	        // Check which specific status changed, prepare code, change state and write new status into the old one.
	        IF (#i_UDT_ArmDiverterStatus.Specific.TimeoutError <> #s_UDT_ArmDiverterOldStatus.Specific.TimeoutError AND NOT #sx_SendAllProcedure)
	            OR (#sx_SendAllProcedure AND #ii_ErrorNumber = 0)
	        THEN
	            #sdi_Code := "DB_MFC_ErrorCode".ArmDiverter.TimeoutError;
	            #si_State := BOOL_TO_INT(#i_UDT_ArmDiverterStatus.Specific.TimeoutError);
	            #s_UDT_ArmDiverterOldStatus.Specific.TimeoutError := #i_UDT_ArmDiverterStatus.Specific.TimeoutError;
	            #sx_ItemErrorMessageReq := TRUE;
	            #ii_ErrorNumber += 1;
	        ELSIF (#i_UDT_ArmDiverterStatus.Specific.LimitHomeError <> #s_UDT_ArmDiverterOldStatus.Specific.LimitHomeError AND NOT #sx_SendAllProcedure)
	            OR (#sx_SendAllProcedure AND #ii_ErrorNumber = 1)
	        THEN
	            #sdi_Code := "DB_MFC_ErrorCode".ArmDiverter.LimitHomeError;
	            #si_State := BOOL_TO_INT(#i_UDT_ArmDiverterStatus.Specific.LimitHomeError);
	            #s_UDT_ArmDiverterOldStatus.Specific.LimitHomeError := #i_UDT_ArmDiverterStatus.Specific.LimitHomeError;
	            #sx_ItemErrorMessageReq := TRUE;
	            #ii_ErrorNumber += 1;
	        ELSIF (#i_UDT_ArmDiverterStatus.Specific.LimitDivertError <> #s_UDT_ArmDiverterOldStatus.Specific.LimitDivertError AND NOT #sx_SendAllProcedure)
	            OR (#sx_SendAllProcedure AND #ii_ErrorNumber = 2)
	        THEN
	            #sdi_Code := "DB_MFC_ErrorCode".ArmDiverter.LimitDivertError;
	            #si_State := BOOL_TO_INT(#i_UDT_ArmDiverterStatus.Specific.LimitDivertError);
	            #s_UDT_ArmDiverterOldStatus.Specific.LimitDivertError := #i_UDT_ArmDiverterStatus.Specific.LimitDivertError;
	            #sx_ItemErrorMessageReq := TRUE;
	            #ii_ErrorNumber += 1;
	        ELSIF (#i_UDT_ArmDiverterStatus.Specific.PXHomeError <> #s_UDT_ArmDiverterOldStatus.Specific.PXHomeError AND NOT #sx_SendAllProcedure)
	            OR (#sx_SendAllProcedure AND #ii_ErrorNumber = 3)
	        THEN
	            #sdi_Code := "DB_MFC_ErrorCode".ArmDiverter.PXHomeError;
	            #si_State := BOOL_TO_INT(#i_UDT_ArmDiverterStatus.Specific.PXHomeError);
	            #s_UDT_ArmDiverterOldStatus.Specific.PXHomeError := #i_UDT_ArmDiverterStatus.Specific.PXHomeError;
	            #sx_ItemErrorMessageReq := TRUE;
	            #ii_ErrorNumber += 1;
	        ELSIF (#i_UDT_ArmDiverterStatus.Specific.PXDivertError <> #s_UDT_ArmDiverterOldStatus.Specific.PXDivertError AND NOT #sx_SendAllProcedure)
	            OR (#sx_SendAllProcedure AND #ii_ErrorNumber = 4)
	        THEN
	            #sdi_Code := "DB_MFC_ErrorCode".ArmDiverter.PXDivertError;
	            #si_State := BOOL_TO_INT(#i_UDT_ArmDiverterStatus.Specific.PXDivertError);
	            #s_UDT_ArmDiverterOldStatus.Specific.PXDivertError := #i_UDT_ArmDiverterStatus.Specific.PXDivertError;
	            #sx_ItemErrorMessageReq := TRUE;
	            #ii_ErrorNumber += 1;
	        ELSIF (#i_UDT_ArmDiverterStatus.Specific.AtHomePosition <> #s_UDT_ArmDiverterOldStatus.Specific.AtHomePosition AND NOT #sx_SendAllProcedure)
	            OR (#sx_SendAllProcedure AND #ii_ErrorNumber = 5)
	        THEN
	            #sdi_Code := "DB_MFC_ErrorCode".ArmDiverter.AtHomePosition;
	            #si_State := BOOL_TO_INT(#i_UDT_ArmDiverterStatus.Specific.AtHomePosition);
	            #s_UDT_ArmDiverterOldStatus.Specific.AtHomePosition := #i_UDT_ArmDiverterStatus.Specific.AtHomePosition;
	            #sx_ItemErrorMessageReq := TRUE;
	            #ii_ErrorNumber += 1;
	        ELSIF (#i_UDT_ArmDiverterStatus.Specific.AtDivertPosition <> #s_UDT_ArmDiverterOldStatus.Specific.AtDivertPosition AND NOT #sx_SendAllProcedure)
	            OR (#sx_SendAllProcedure AND #ii_ErrorNumber = 6)
	        THEN
	            #sdi_Code := "DB_MFC_ErrorCode".ArmDiverter.AtDivertPosition;
	            #si_State := BOOL_TO_INT(#i_UDT_ArmDiverterStatus.Specific.AtDivertPosition);
	            #s_UDT_ArmDiverterOldStatus.Specific.AtDivertPosition := #i_UDT_ArmDiverterStatus.Specific.AtDivertPosition;
	            #sx_ItemErrorMessageReq := TRUE;
	            #ii_ErrorNumber += 1;
	        ELSIF (#i_UDT_ArmDiverterStatus.Specific.ReferencError <> #s_UDT_ArmDiverterOldStatus.Specific.ReferencError AND NOT #sx_SendAllProcedure)
	            OR (#sx_SendAllProcedure AND #ii_ErrorNumber = 7)
	        THEN
	            #sdi_Code := "DB_MFC_ErrorCode".ArmDiverter.ReferencError;
	            #si_State := BOOL_TO_INT(#i_UDT_ArmDiverterStatus.Specific.ReferencError);
	            #s_UDT_ArmDiverterOldStatus.Specific.ReferencError := #i_UDT_ArmDiverterStatus.Specific.ReferencError;
	            #sx_ItemErrorMessageReq := TRUE;
	            #ii_ErrorNumber += 1;
	        ELSIF (#i_UDT_ArmDiverterStatus.Specific.ParcelDivertError <> #s_UDT_ArmDiverterOldStatus.Specific.ParcelDivertError AND NOT #sx_SendAllProcedure)
	            OR (#sx_SendAllProcedure AND #ii_ErrorNumber = 8)
	        THEN
	            #sdi_Code := "DB_MFC_ErrorCode".ArmDiverter.ParcelDivertError;
	            #si_State := BOOL_TO_INT(#i_UDT_ArmDiverterStatus.Specific.ParcelDivertError);
	            #s_UDT_ArmDiverterOldStatus.Specific.ParcelDivertError := #i_UDT_ArmDiverterStatus.Specific.ParcelDivertError;
	            #sx_ItemErrorMessageReq := TRUE;
	            #sx_SendAllProcedure := FALSE;
	        END_IF;
	    END_IF;
	END_REGION

	REGION 4 - Write message components to the item error structure

	    #s_UDT_ItemError.ItemNumber := #i_UDT_EquipmentNumber;
	    #s_UDT_ItemError.Error := #sdi_Code;
	    #s_UDT_ItemError.State := #si_State;
	    #s_UDT_ItemError.Masked := 1;

	END_REGION

	REGION 5 - Write message components to the item status structure

	    #s_UDT_ItemStatus.Group := #i_UDT_EquipmentNumber.Group;
	    #s_UDT_ItemStatus.Node := #i_UDT_EquipmentNumber.Node;
	    #s_UDT_ItemStatus.Status := #si_ItemStatus;

	END_REGION

	REGION 6 - Prepare messages to the MFC

	    // If item error message required signal is set, prepare the item error message.
	    IF (#sx_ItemErrorMessageReq)
	    THEN
	        #s_FB_ItemError(i_UDT_ItemErrorBody := #s_UDT_ItemError,
	                        ii_MessageGroup := 1,
	                        ix_FlagRetry := FALSE,
	                        idi_TimeSpan := 0,
	                        qx_Error => #sx_ItemErrorBlockError,
	                        qx_Warning => #sx_ItemErrorBlockWarning,
	                        iq_UDT_FifoHeader := #iq_UDT_FifoHeader,
	                        iqs_FifoData := #iqs_FifoData,
	                        iqdi_MessageSequenceNumber := #iqdi_MessageSequenceNumber);
	    END_IF;

	    // If item status message required signal is set, prepare the item error message.
	    IF (#sx_ItemStatusMessageReq)
	    THEN
	        #s_FB_ItemStatus(i_UDT_ItemStatusBody := #s_UDT_ItemStatus,
	                         ii_MessageGroup := 1,
	                         ix_FlagRetry := FALSE,
	                         idi_TimeSpan := 0,
	                         qx_Error => #sx_ItemStatusBlockError,
	                         qx_Warning => #sx_ItemStatusBlockWarning,
	                         iq_UDT_FifoHeader := #iq_UDT_FifoHeader,
	                         iqs_FifoData := #iqs_FifoData,
	                         iqdi_MessageSequenceNumber := #iqdi_MessageSequenceNumber);
	    END_IF;

	END_REGION

	REGION 7 - Write outputs

	    // Prepare collective output error.
	    #qx_Error :=
	    #sx_ItemErrorBlockError
	    OR #sx_ItemStatusBlockError
	    OR #sx_FIFOError;

	    // Prepare collective output warning.
	    #qx_Warning :=
	    #sx_ItemErrorBlockWarning
	    OR #sx_ItemStatusBlockWarning
	    OR #sx_FIFOWarning;

	END_REGION




END_FUNCTION_BLOCK

FUNCTION_BLOCK "FB_MFC_Visu_TCPIPSend"
TITLE = FB_TCPIPSend
{ S7_Optimized_Access := 'TRUE' }
AUTHOR : MHSE
FAMILY : Communication
VERSION : 2.0
// ATTRIBUTES
// AUTO_NUMBER = True
// BLOCK_NUMBER = 162
// END_ATTRIBUTES
//Function block to send data from TCPIP.
   VAR_INPUT
      i_UDT_Connection { ExternalAccessible := 'False'; ExternalVisible := 'False'; ExternalWritable := 'False'} : "UDT_Connection";   // Connection parameters
      ii_HeaderLength { ExternalAccessible := 'False'; ExternalVisible := 'False'; ExternalWritable := 'False'} : Int;   // Message header length
      ii_BodyLengthPosition { ExternalAccessible := 'False'; ExternalVisible := 'False'; ExternalWritable := 'False'} : Int;   // Position in header where message body length value starts
      ix_EnableSend { ExternalAccessible := 'False'; ExternalVisible := 'False'; ExternalWritable := 'False'} : Bool;   // TRUE when send is enable
   END_VAR

   VAR_OUTPUT
      qx_Error { ExternalAccessible := 'False'; ExternalVisible := 'False'; ExternalWritable := 'False'} : Bool;   // TRUE when collective block error occurred
      qx_Warning { ExternalAccessible := 'False'; ExternalVisible := 'False'; ExternalWritable := 'False'} : Bool;   // TRUE when collective block warning occurred
   END_VAR

   VAR_IN_OUT
      iq_UDT_FifoLowHeader : "UDT_FifoHeader";   // Low priority FIFO header
      iqs_FifoLowData : Variant;   // Low priority FIFO data
      iq_UDT_FifoMediumHeader : "UDT_FifoHeader";   // Medium priority FIFO header
      iqs_FifoMediumData : Variant;   // Medium priority FIFO data
      iq_UDT_FifoHighHeader : "UDT_FifoHeader";   // High priority FIFO header
      iqs_FifoHighData : Variant;   // High priority FIFO data
   END_VAR

   VAR
      s_FB_TSEND {InstructionName := 'TSEND'; LibVersion := '4.0'; ExternalAccessible := 'False'; ExternalVisible := 'False'; ExternalWritable := 'False'; S7_SetPoint := 'False'} : TSEND;   // Siemens "TSEND" block - to send the data over TCPIP socket
      s_UDT_MessageArray { ExternalAccessible := 'False'; ExternalVisible := 'False'; ExternalWritable := 'False'; S7_SetPoint := 'False'} : "UDT_MessageV2";   // Message
      ss_TSEND { ExternalAccessible := 'False'; ExternalVisible := 'False'; ExternalWritable := 'False'} : Struct   // TSEND block structure
         Status { ExternalAccessible := 'False'; ExternalVisible := 'False'; ExternalWritable := 'False'} : Word;   //    TSEND - Status
         Request { ExternalAccessible := 'False'; ExternalVisible := 'False'; ExternalWritable := 'False'} : Bool;   //    TSEND - Request
         Busy { ExternalAccessible := 'False'; ExternalVisible := 'False'; ExternalWritable := 'False'} : Bool;   //    TSEND - Busy
         Done { ExternalAccessible := 'False'; ExternalVisible := 'False'; ExternalWritable := 'False'} : Bool;   //    TSEND - Done
         Error { ExternalAccessible := 'False'; ExternalVisible := 'False'; ExternalWritable := 'False'} : Bool;   //    TSEND - Error
      END_STRUCT;
      ss_Status { ExternalAccessible := 'False'; ExternalVisible := 'False'; ExternalWritable := 'False'} : Struct   // Status structure
         FIFOLowPriorityStatus { ExternalAccessible := 'False'; ExternalVisible := 'False'; ExternalWritable := 'False'} : "UDT_FifoStatus";
         FIFOMedPriorityStatus { ExternalAccessible := 'False'; ExternalVisible := 'False'; ExternalWritable := 'False'} : "UDT_FifoStatus";
         FIFOHighPriorityStatus { ExternalAccessible := 'False'; ExternalVisible := 'False'; ExternalWritable := 'False'} : "UDT_FifoStatus";
         FIFOLowPriorityError { ExternalAccessible := 'False'; ExternalVisible := 'False'; ExternalWritable := 'False'} : Bool;   // FIFO low priority error
         FIFOLowPriorityWarning { ExternalAccessible := 'False'; ExternalVisible := 'False'; ExternalWritable := 'False'} : Bool;   // FIFO low priority warning
         FIFOMedPriorityError { ExternalAccessible := 'False'; ExternalVisible := 'False'; ExternalWritable := 'False'} : Bool;   // FIFO medium priority error
         FIFOMedPriorityWarning { ExternalAccessible := 'False'; ExternalVisible := 'False'; ExternalWritable := 'False'} : Bool;   // FIFO medium priority warning
         FIFOHighPriorityError { ExternalAccessible := 'False'; ExternalVisible := 'False'; ExternalWritable := 'False'} : Bool;   // FIFO high priority error
         FIFOHighPriorityWarning { ExternalAccessible := 'False'; ExternalVisible := 'False'; ExternalWritable := 'False'} : Bool;   // FIFO high priority warning
         SendError { ExternalAccessible := 'False'; ExternalVisible := 'False'; ExternalWritable := 'False'} : Bool;   // Send operation error
      END_STRUCT;
      sw_BodyLength { ExternalAccessible := 'False'; ExternalVisible := 'False'; ExternalWritable := 'False'} : Word;   // Message body length
      si_MessageLength { ExternalAccessible := 'False'; ExternalVisible := 'False'; ExternalWritable := 'False'} : Int;   // Message length
      sx_MessageReady { ExternalAccessible := 'False'; ExternalVisible := 'False'; ExternalWritable := 'False'} : Bool;   // Message is ready to send
      sx_MessageRead { ExternalAccessible := 'False'; ExternalVisible := 'False'; ExternalWritable := 'False'} : Bool;   // Message has been read
      sx_MessageReadRequest { ExternalAccessible := 'False'; ExternalVisible := 'False'; ExternalWritable := 'False'} : Bool;   // Request to read message
      sx_FIFOError { ExternalAccessible := 'False'; ExternalVisible := 'False'; ExternalWritable := 'False'} : Bool;   // Summary FIFO error
   END_VAR


BEGIN
	(*
	----------------------------------------------------------------------------------------
	|                                                                                      |
	|  Copyright  2023             FORTNA Europe BV                                        |
	|  All Rights Reserved         Netherlands                                             |
	|                                                                                      |
	----------------------------------------------------------------------------------------
	Version history:
	Date        | Version   | Author       | Remark
	----------------------------------------------------------------------------------------
	24/10/2019  | 3.0       | L.Klar       | Initial version
	12/03/2020  | 3.1       | M.Kurpiers   | Adapting reviews
	16/01/2023  | 4.0       | S. Nikodem   | Release TIA 17 | DHL Munich 2023
	13/03/2023  | 4.1       | S. Nieswiec  | Updated for new Baseline
	*)

	REGION 1 – Update FIFO header status bits

	    // Mode 'S' - High priority FIFO register status update.
	    "FC_Fifo"(ic_Mode := 'S',
	              qUDT_Status => #ss_Status.FIFOHighPriorityStatus,
	              qx_Error => #ss_Status.FIFOHighPriorityError,
	              qx_Warning => #ss_Status.FIFOHighPriorityWarning,
	              iqv_Data := #s_UDT_MessageArray,
	              iqUDT_FifoHeader := #iq_UDT_FifoHighHeader,
	              iqv_DataBuffer := #iqs_FifoHighData);

	    // Mode 'S' - Medium priority FIFO register status update.
	    "FC_Fifo"(ic_Mode := 'S',
	              qUDT_Status => #ss_Status.FIFOMedPriorityStatus,
	              qx_Error => #ss_Status.FIFOMedPriorityError,
	              qx_Warning => #ss_Status.FIFOMedPriorityWarning,
	              iqv_Data := #s_UDT_MessageArray,
	              iqUDT_FifoHeader := #iq_UDT_FifoMediumHeader,
	              iqv_DataBuffer := #iqs_FifoMediumData);

	    // Mode 'S' - Low priority FIFO register status update.
	    "FC_Fifo"(ic_Mode := 'S',
	              qUDT_Status => #ss_Status.FIFOLowPriorityStatus,
	              qx_Error => #ss_Status.FIFOLowPriorityError,
	              qx_Warning => #ss_Status.FIFOLowPriorityWarning,
	              iqv_Data := #s_UDT_MessageArray,
	              iqUDT_FifoHeader := #iq_UDT_FifoLowHeader,
	              iqv_DataBuffer := #iqs_FifoLowData);

	END_REGION

	REGION 2 – FIFO header summary error

	    #sx_FIFOError :=
	    #ss_Status.FIFOHighPriorityError
	    OR #ss_Status.FIFOMedPriorityError
	    OR #ss_Status.FIFOLowPriorityError;

	END_REGION

	REGION 3 – FIFO Read request

	    #sx_MessageReadRequest :=
	    #ix_EnableSend
	    AND NOT #sx_FIFOError
	    AND NOT #ss_TSEND.Error
	    AND #ss_TSEND.Status = 16#7000;

	END_REGION

	REGION 4 – Read the message from high priority FIFO data buffer

	    IF #sx_MessageReadRequest
	        AND NOT #iq_UDT_FifoHighHeader.Status.Empty
	        AND NOT #sx_MessageRead
	    THEN
	        // Mode 'R' - Read high priority FIFO record.
	        "FC_Fifo"(ic_Mode := 'R',
	                  qUDT_Status => #ss_Status.FIFOHighPriorityStatus,
	                  qx_Error => #ss_Status.FIFOHighPriorityError,
	                  qx_Warning => #ss_Status.FIFOHighPriorityWarning,
	                  iqv_Data := #s_UDT_MessageArray,
	                  iqUDT_FifoHeader := #iq_UDT_FifoHighHeader,
	                  iqv_DataBuffer := #iqs_FifoHighData);

	        #sx_MessageRead := TRUE;
	    END_IF;

	END_REGION

	REGION 5 – Read the message from medium priority FIFO data buffer

	    IF #sx_MessageReadRequest
	        AND #iq_UDT_FifoHighHeader.Status.Empty
	        AND NOT #iq_UDT_FifoMediumHeader.Status.Empty
	        AND NOT #sx_MessageRead
	    THEN
	        // Mode 'R' - Read medium priority FIFO record.
	        "FC_Fifo"(ic_Mode := 'R',
	                  qUDT_Status => #ss_Status.FIFOMedPriorityStatus,
	                  qx_Error => #ss_Status.FIFOMedPriorityError,
	                  qx_Warning => #ss_Status.FIFOMedPriorityWarning,
	                  iqv_Data := #s_UDT_MessageArray,
	                  iqUDT_FifoHeader := #iq_UDT_FifoMediumHeader,
	                  iqv_DataBuffer := #iqs_FifoMediumData);

	        #sx_MessageRead := TRUE;
	    END_IF;

	END_REGION

	REGION 6 – Read the message from low priority FIFO data buffer

	    IF #sx_MessageReadRequest
	        AND #iq_UDT_FifoHighHeader.Status.Empty
	        AND #iq_UDT_FifoMediumHeader.Status.Empty
	        AND NOT #iq_UDT_FifoLowHeader.Status.Empty
	        AND NOT #sx_MessageRead
	    THEN
	        #sx_MessageRead := TRUE;

	        // Mode 'R' - Read low priority FIFO record.
	        "FC_Fifo"(ic_Mode := 'R',
	                  qUDT_Status => #ss_Status.FIFOLowPriorityStatus,
	                  qx_Error => #ss_Status.FIFOLowPriorityError,
	                  qx_Warning => #ss_Status.FIFOLowPriorityWarning,
	                  iqv_Data := #s_UDT_MessageArray,
	                  iqUDT_FifoHeader := #iq_UDT_FifoLowHeader,
	                  iqv_DataBuffer := #iqs_FifoLowData);
	    END_IF;

	END_REGION

	REGION 7 – Message length

	    // Measuring the length of a read message.
	    IF #sx_MessageRead
	        AND NOT #sx_MessageReady
	    THEN
	        // Initialize the message length.
	        #si_MessageLength := 0;

	        // Get the length of the message by extracting the body length from the message header.
	        #sw_BodyLength := #s_UDT_MessageArray.Bytes[#ii_BodyLengthPosition];
	        #si_MessageLength := WORD_TO_INT(IN := SHL(IN := #sw_BodyLength, N := 8)) + BYTE_TO_INT(#s_UDT_MessageArray.Bytes[#ii_BodyLengthPosition + 1]) + #ii_HeaderLength;
	        #sx_MessageReady := TRUE;
	    END_IF;

	END_REGION

	REGION 8 – Send request

	    IF #sx_MessageRead
	        AND #sx_MessageReady
	    THEN
	        #ss_TSEND.Request := TRUE;
	    END_IF;

	END_REGION

	REGION 9 – Send data

	    #s_FB_TSEND(REQ := #ss_TSEND.Request,
	                ID := #i_UDT_Connection.ID,
	                LEN := INT_TO_UDINT(#si_MessageLength),
	                DONE => #ss_TSEND.Done,
	                BUSY => #ss_TSEND.Busy,
	                ERROR => #ss_TSEND.Error,
	                STATUS => #ss_TSEND.Status,
	                DATA := #s_UDT_MessageArray);

	    // Reset send request, message read and ready bits.
	    IF #ss_TSEND.Request
	        AND NOT #ss_TSEND.Busy
	        AND (#ss_TSEND.Done
	        OR #ss_TSEND.Status = 16#7000)
	    THEN
	        #ss_TSEND.Request := FALSE;
	        #sx_MessageRead := FALSE;
	        #sx_MessageReady := FALSE;
	    END_IF;

	    // Reset send error and TSEND status after correctly sent message.
	    IF #ss_TSEND.Done
	    THEN
	        #ss_Status.SendError := FALSE;
	    END_IF;

	    // Set send error and TSEND status if error occured.
	    IF #ss_TSEND.Error
	    THEN
	        #ss_Status.SendError := TRUE;
	    END_IF;

	END_REGION

	REGION 10 – Status

	    // Parametrization collective error output.
	    #qx_Error :=
	    #sx_FIFOError
	    OR #ss_Status.SendError;

	    // Parametrization collective warning output.
	    #qx_Warning :=
	    #ss_Status.FIFOHighPriorityWarning
	    OR #ss_Status.FIFOMedPriorityWarning
	    OR #ss_Status.FIFOLowPriorityWarning;

	END_REGION
END_FUNCTION_BLOCK

FUNCTION_BLOCK "FB_MFC_Visu_Conveyor_Status"
{ S7_Optimized_Access := 'TRUE' }
VERSION : 0.1
// ATTRIBUTES
// AUTO_NUMBER = True
// BLOCK_NUMBER = 141
// END_ATTRIBUTES
   VAR_INPUT
      ix_SendAllErrorsState { ExternalAccessible := 'False'; ExternalVisible := 'False'; ExternalWritable := 'False'} : Bool;   // True - update all the messages
      ix_MFCConnected { ExternalAccessible := 'False'; ExternalVisible := 'False'; ExternalWritable := 'False'} : Bool;   // True - A connection to the MFC has been established
      ix_CollectiveReset { ExternalAccessible := 'False'; ExternalVisible := 'False'; ExternalWritable := 'False'} : Bool;   // True - Collective reset command of all system controls
      i_UDT_MaintenanceCounterConfiguration { ExternalAccessible := 'False'; ExternalVisible := 'False'; ExternalWritable := 'False'} : "UDT_MaintenanceCounterConfiguration" := (86400, 10000000, 100);   // Maintenance counter configuration
      i_UDT_ConveyorInterface { ExternalAccessible := 'False'; ExternalVisible := 'False'; ExternalWritable := 'False'} : "UDT_ConveyorInterface";   // Input conveyor interface structrue
      i_UDT_ConveyorStatus { ExternalAccessible := 'False'; ExternalVisible := 'False'; ExternalWritable := 'False'} : "UDT_ConveyorStatus";   // Input Conveyor status structure
      i_UDT_EquipmentNumber { ExternalAccessible := 'False'; ExternalVisible := 'False'; ExternalWritable := 'False'} : "UDT_EquipmentNumber";   // Item number
   END_VAR

   VAR_OUTPUT
      qx_Error { ExternalAccessible := 'False'; ExternalVisible := 'False'; ExternalWritable := 'False'} : Bool;   // Block error
      qx_Warning { ExternalAccessible := 'False'; ExternalVisible := 'False'; ExternalWritable := 'False'} : Bool;   // Block warning
   END_VAR

   VAR_IN_OUT
      iq_UDT_FifoHeader : "UDT_FifoHeader";   // FIFO header
      iqs_FifoData : Array[*] of "UDT_MessageV2";   // FIFO data buffer
      iqdi_MessageSequenceNumber { ExternalAccessible := 'False'; ExternalVisible := 'False'; ExternalWritable := 'False'} : DInt;   // Message number
   END_VAR

   VAR
      s_FB_ItemError { ExternalAccessible := 'False'; ExternalVisible := 'False'; ExternalWritable := 'False'; S7_SetPoint := 'False'} : "FB_ItemError";   // Item error block's instance
      s_FB_ItemStatus { ExternalAccessible := 'False'; ExternalVisible := 'False'; ExternalWritable := 'False'; S7_SetPoint := 'False'} : "FB_ItemStatus";   // Item status block's instance
      s_FB_MaintenanceCounter { ExternalAccessible := 'False'; ExternalVisible := 'False'; ExternalWritable := 'False'; S7_SetPoint := 'False'} : "FB_MaintenanceCounter";   // Maintenence counter message block instance
      s_UDT_ItemError { ExternalAccessible := 'False'; ExternalVisible := 'False'; ExternalWritable := 'False'; S7_SetPoint := 'False'} : "UDT_ItemError";   // Item error message body structure
      s_UDT_ItemStatus { ExternalAccessible := 'False'; ExternalVisible := 'False'; ExternalWritable := 'False'; S7_SetPoint := 'False'} : "UDT_ItemStatus";   // Item status message body structure
      s_UDT_Message { ExternalAccessible := 'False'; ExternalVisible := 'False'; ExternalWritable := 'False'; S7_SetPoint := 'False'} : "UDT_BytesMessage";   // Message
      s_UDT_ConveyorOld { ExternalAccessible := 'False'; ExternalVisible := 'False'; ExternalWritable := 'False'; S7_SetPoint := 'False'} : "UDT_ConveyorStatus";   // Conveyor old status structure
      s_UDT_ConveyorInterfaceOld { ExternalAccessible := 'False'; ExternalVisible := 'False'; ExternalWritable := 'False'; S7_SetPoint := 'False'} : "UDT_ConveyorInterface";   // Conveyor old interface structure
      s_UDT_FIFOStatus { ExternalAccessible := 'False'; ExternalVisible := 'False'; ExternalWritable := 'False'; S7_SetPoint := 'False'} : "UDT_FifoStatus";   // FIFO status structure
      ss_FIFOStatus { ExternalAccessible := 'False'; ExternalVisible := 'False'; ExternalWritable := 'False'; S7_SetPoint := 'False'} : "UDT_FifoStatus";   // Status structure
      s_R_TRIG_ConveyorStart {InstructionName := 'R_TRIG'; LibVersion := '1.0'; ExternalAccessible := 'False'; ExternalVisible := 'False'; ExternalWritable := 'False'; S7_SetPoint := 'False'} : R_TRIG;   // Rising edge trigger Conveyor start
      s_R_TRIG_Connection {InstructionName := 'R_TRIG'; LibVersion := '1.0'; ExternalAccessible := 'False'; ExternalVisible := 'False'; ExternalWritable := 'False'; S7_SetPoint := 'False'} : R_TRIG;   // Rising edge trigger connection reastablished
      s_F_TRIG_ConveyorStop {InstructionName := 'F_TRIG'; LibVersion := '1.0'; ExternalAccessible := 'False'; ExternalVisible := 'False'; ExternalWritable := 'False'; S7_SetPoint := 'False'} : F_TRIG;   // Falling edge trigger Conveyor stop
      s_F_TRIG_SendAllErrors {InstructionName := 'F_TRIG'; LibVersion := '1.0'; ExternalAccessible := 'False'; ExternalVisible := 'False'; ExternalWritable := 'False'; S7_SetPoint := 'False'} : F_TRIG;   // Falling edge trigger from signal send all errors
      slr_RunningTimeMS { ExternalAccessible := 'False'; ExternalVisible := 'False'; ExternalWritable := 'False'} : LReal;   // Conveyor running time [ms]
      sdi_DistanceTraveled { ExternalAccessible := 'False'; ExternalVisible := 'False'; ExternalWritable := 'False'} : DInt;   // Distance traveled by conveyor
      sdi_StartStop { ExternalAccessible := 'False'; ExternalVisible := 'False'; ExternalWritable := 'False'} : DInt;   // Value of change conveyor state from start to stop and from stop to start
      sdi_Code { ExternalAccessible := 'False'; ExternalVisible := 'False'; ExternalWritable := 'False'} : DInt;   // Error code
      sdi_RunningTime { ExternalAccessible := 'False'; ExternalVisible := 'False'; ExternalWritable := 'False'} : DInt;   // Conveyor running time [s]
      si_ItemStatus { ExternalAccessible := 'False'; ExternalVisible := 'False'; ExternalWritable := 'False'} : Int;   // Item status
      si_State { ExternalAccessible := 'False'; ExternalVisible := 'False'; ExternalWritable := 'False'} : Int;   // Error state
      ii_ErrorNumber { ExternalAccessible := 'False'; ExternalVisible := 'False'; ExternalWritable := 'False'} : Int;   // Counter Error Number
      sx_ItemErrorMessageReq { ExternalAccessible := 'False'; ExternalVisible := 'False'; ExternalWritable := 'False'} : Bool;   // Item error message required
      sx_ItemStatusMessageReq { ExternalAccessible := 'False'; ExternalVisible := 'False'; ExternalWritable := 'False'} : Bool;   // Item status message required
      sx_ItemErrorBlockError { ExternalAccessible := 'False'; ExternalVisible := 'False'; ExternalWritable := 'False'} : Bool;   // Item error block error
      sx_ItemStatusBlockError { ExternalAccessible := 'False'; ExternalVisible := 'False'; ExternalWritable := 'False'} : Bool;   // Item status block error
      sx_FIFOError { ExternalAccessible := 'False'; ExternalVisible := 'False'; ExternalWritable := 'False'} : Bool;   // FIFO error
      sx_FIFOWarning { ExternalAccessible := 'False'; ExternalVisible := 'False'; ExternalWritable := 'False'} : Bool;   // FIFO warning
      sx_MaintenanceCounterBlockError { ExternalAccessible := 'False'; ExternalVisible := 'False'; ExternalWritable := 'False'} : Bool;   // Maintenance counter block error
      sx_ItemStatusBlockWarning { ExternalAccessible := 'False'; ExternalVisible := 'False'; ExternalWritable := 'False'} : Bool;   // Item status block warning
      sx_ItemErrorBlockWarning { ExternalAccessible := 'False'; ExternalVisible := 'False'; ExternalWritable := 'False'} : Bool;   // Item error block warning
      sx_MaintenanceCounterBlockWarning { ExternalAccessible := 'False'; ExternalVisible := 'False'; ExternalWritable := 'False'} : Bool;   // Maintenance counter block warning
      sx_SendAllProcedure { ExternalAccessible := 'False'; ExternalVisible := 'False'; ExternalWritable := 'False'} : Bool;   // Send all procedure
   END_VAR

   VAR CONSTANT
      ci_MessageGroup : Int := 1;
      ci_TimeSpan : Int := 0;
   END_VAR


BEGIN
	(*
	----------------------------------------------------------------------------------------
	|                                                                                      |
	|  Copyright  2023             FORTNA Europe BV                                        |
	|  All Rights Reserved         Netherlands                                             |
	|                                                                                      |
	----------------------------------------------------------------------------------------
	Version history:
	Date        | Version   | Author       | Remark
	----------------------------------------------------------------------------------------
	03/01/2023  | 1.0       | S. Nikodem   | Release TIA 17 | DHL Munich 2023
	09/08/2023  | 2.0       | S. Theocharis| Update with DB error code | DHL Munich 2023
	13/03/2023  | 2.1       | S. Nieswiec  | Updated for new Baseline

	*)

	REGION 1 - Initialize message required signals

	    #sx_ItemErrorMessageReq := FALSE;
	    #sx_ItemStatusMessageReq := FALSE;

	    // On connection reestablish send last remembered status and error state ( status only when it's diffrent then 0 )
	    #s_R_TRIG_Connection(CLK := #ix_MFCConnected);

	    // IF #s_R_TRIG_Connection.Q AND #si_ItemStatus <> 0
	    // THEN
	    //     #ii_ErrorNumber := 0;
	    //     #sx_SendAllProcedure := TRUE;
	    //    // #sx_ItemStatusMessageReq := TRUE;
	    // END_IF;

	    // IF #s_R_TRIG_Connection.Q
	    // THEN
	    //     #ii_ErrorNumber := 0;
	    //     #sx_SendAllProcedure := TRUE;
	    //    // #sx_ItemErrorMessageReq := TRUE;
	    // END_IF;

	    // Prepare trigger on the collective reset signal.
	    #s_F_TRIG_SendAllErrors(CLK := #ix_SendAllErrorsState);

	    // When collective reset will go down, start send every equipment errors.
	    IF #s_F_TRIG_SendAllErrors.Q AND NOT #sx_SendAllProcedure
	    THEN
	        #ii_ErrorNumber := 0;
	        #sx_SendAllProcedure := TRUE;
	    END_IF;

	END_REGION

	REGION 2 - O header status update

	    // Mode 'S' - FIFO register status update.
	    "FC_Fifo"(ic_Mode := 'S',
	              qUDT_Status => #ss_FIFOStatus,
	              qx_Error => #sx_FIFOError,
	              qx_Warning => #sx_FIFOWarning,
	              iqv_Data := #s_UDT_Message,
	              iqUDT_FifoHeader := #iq_UDT_FifoHeader,
	              iqv_DataBuffer := #iqs_FifoData);

	END_REGION

	REGION 2 - Prepare message data

	    // When there is no reset errors command, update status and errors.
	    IF NOT #ix_CollectiveReset
	        AND NOT #ss_FIFOStatus.FifoPreFull
	    THEN

	        IF (#i_UDT_ConveyorStatus.Status <> #s_UDT_ConveyorOld.Status OR (#sx_SendAllProcedure AND #ii_ErrorNumber = 0))
	        THEN
	            #sx_ItemStatusMessageReq := TRUE;
	            #si_ItemStatus := #i_UDT_ConveyorStatus.Status;
	            #s_UDT_ConveyorOld.Status := #i_UDT_ConveyorStatus.Status;
	        END_IF;

	        // Check which specific status changed, prepare code, change state and write new status into the old one.
	        (*
	       // Do not send the internal tracking error / / internal tracking warning
	        IF (#i_UDT_ConveyorInterface.InternalErrorTracking <> #s_UDT_ConveyorInterfaceOld.InternalErrorTracking AND NOT #sx_SendAllProcedure)
	            OR (#sx_SendAllProcedure AND #ii_ErrorNumber = 0)

	        THEN
	            #sdi_Code := "DB_MFC_ErrorCode".ConveyorInterface.InternalErrorTracking;
	            #si_State := BOOL_TO_INT(#i_UDT_ConveyorInterface.InternalErrorTracking);
	            #s_UDT_ConveyorInterfaceOld.InternalErrorTracking := #i_UDT_ConveyorInterface.InternalErrorTracking;
	            #sx_ItemErrorMessageReq := TRUE;
	            // #qw_AlarmWord1.%X0 := #s_UDT_ConveyorInterface.InternalErrorTracking;
	            #ii_ErrorNumber += 1;
	        ELSIF (#i_UDT_ConveyorInterface.InternalWarningTracking <> #s_UDT_ConveyorInterfaceOld.InternalWarningTracking AND NOT #sx_SendAllProcedure)
	            OR (#sx_SendAllProcedure AND #ii_ErrorNumber = 1)
	        THEN
	            #sdi_Code := "DB_MFC_ErrorCode".ConveyorInterface.InternalWarningTracking;
	            #si_State := BOOL_TO_INT(#i_UDT_ConveyorInterface.InternalWarningTracking);
	            #s_UDT_ConveyorInterfaceOld.InternalWarningTracking := #i_UDT_ConveyorInterface.InternalWarningTracking;
	            #sx_ItemErrorMessageReq := TRUE;
	            //  #qw_AlarmWord1.%X1 := #s_UDT_ConveyorInterface.InternalWarningTracking;
	            #ii_ErrorNumber += 1;

	        ELSIF (#i_UDT_ConveyorInterface.Disconnected <> #s_UDT_ConveyorInterfaceOld.Disconnected AND NOT #sx_SendAllProcedure)
	            OR (#sx_SendAllProcedure AND #ii_ErrorNumber = 2)
	        *)
	        IF (#i_UDT_ConveyorInterface.Disconnected <> #s_UDT_ConveyorInterfaceOld.Disconnected AND NOT #sx_SendAllProcedure)
	            OR (#sx_SendAllProcedure AND #ii_ErrorNumber = 0)

	        THEN
	            #sdi_Code := "DB_MFC_ErrorCode".ConveyorInterface.Disconnected;
	            #si_State := BOOL_TO_INT(#i_UDT_ConveyorInterface.Disconnected);
	            #s_UDT_ConveyorInterfaceOld.Disconnected := #i_UDT_ConveyorInterface.Disconnected;
	            #sx_ItemErrorMessageReq := TRUE;
	            // #qw_AlarmWord1.%X2 := #s_UDT_ConveyorInterface.Disconnected;
	            #sx_SendAllProcedure := FALSE;

	        END_IF;

	    END_IF;

	END_REGION

	REGION 3 - Write message components to the item error structure

	    #s_UDT_ItemError.ItemNumber := #i_UDT_EquipmentNumber;
	    #s_UDT_ItemError.Error := #sdi_Code;
	    #s_UDT_ItemError.State := #si_State;
	    #s_UDT_ItemError.Masked := 1;

	END_REGION

	REGION 4 - Write message components to the item status structure


	    #s_UDT_ItemStatus.Group := #i_UDT_EquipmentNumber.Group;
	    #s_UDT_ItemStatus.Node := #i_UDT_EquipmentNumber.Node;
	    #s_UDT_ItemStatus.Status := #si_ItemStatus;

	END_REGION

	REGION 5 - Prepare messages to the MFC

	    // If item error message required signal is set, prepare the item error message.
	    IF (#sx_ItemErrorMessageReq)
	    THEN
	        #s_FB_ItemError(i_UDT_ItemErrorBody := #s_UDT_ItemError,
	                        ii_MessageGroup := #ci_MessageGroup,
	                        ix_FlagRetry := FALSE,
	                        idi_TimeSpan := #ci_TimeSpan,
	                        qx_Error => #sx_ItemErrorBlockError,
	                        qx_Warning => #sx_ItemErrorBlockWarning,
	                        iq_UDT_FifoHeader := #iq_UDT_FifoHeader,
	                        iqs_FifoData := #iqs_FifoData,
	                        iqdi_MessageSequenceNumber := #iqdi_MessageSequenceNumber);
	    END_IF;

	    // If item status message required signal is set, prepare the item error message.
	    IF (#sx_ItemStatusMessageReq)
	    THEN
	        #s_FB_ItemStatus(i_UDT_ItemStatusBody := #s_UDT_ItemStatus,
	                         ii_MessageGroup := #ci_MessageGroup,
	                         ix_FlagRetry := FALSE,
	                         idi_TimeSpan := #ci_TimeSpan,
	                         qx_Error => #sx_ItemStatusBlockError,
	                         qx_Warning => #sx_ItemStatusBlockWarning,
	                         iq_UDT_FifoHeader := #iq_UDT_FifoHeader,
	                         iqs_FifoData := #iqs_FifoData,
	                         iqdi_MessageSequenceNumber := #iqdi_MessageSequenceNumber);
	    END_IF;

	END_REGION

	REGION 6 - Maintenance counter message

	    // Maintenance counter message is used to inform the MFC about one of three values. When one of them exceed the configured one, message is prepared and sent.
	    // Values which program is counting :
	    // - distance traveled by conveyor,
	    // - change the state of the conveyor ( stop --> start and start --> stop)
	    // - running time of the conveyor.

	    // Calculate conveyor traveled distance.
	    #sdi_DistanceTraveled += #i_UDT_ConveyorInterface.Displacement * 10;

	    // Calculate start-stop.
	    #s_R_TRIG_ConveyorStart(CLK := #i_UDT_ConveyorInterface.RunFwd OR #i_UDT_ConveyorInterface.RunRvs);
	    #s_F_TRIG_ConveyorStop(CLK := #i_UDT_ConveyorInterface.RunRvs OR #i_UDT_ConveyorInterface.RunFwd);

	    // Increment counter on the change of the conveyor's state.
	    IF #s_R_TRIG_ConveyorStart.Q
	        OR #s_F_TRIG_ConveyorStop.Q
	    THEN
	        #sdi_StartStop += 1;
	    END_IF;

	    // Calculate running time.
	    IF #i_UDT_ConveyorInterface.RunFwd
	        OR #i_UDT_ConveyorInterface.RunRvs
	    THEN
	        #slr_RunningTimeMS += "DB_Memory".PrevCycleTime;

	        IF #slr_RunningTimeMS >= 1000
	        THEN
	            #sdi_RunningTime += 1;
	            #slr_RunningTimeMS -= 1000;
	        END_IF;

	    END_IF;

	    // Prepare the maintenance counter message when one of the counted values is equal or bigger then configured one.
	    IF #sdi_RunningTime >= #i_UDT_MaintenanceCounterConfiguration.RunningTime
	        OR #sdi_DistanceTraveled >= #i_UDT_MaintenanceCounterConfiguration.DistanceTraveled
	        OR #sdi_StartStop >= #i_UDT_MaintenanceCounterConfiguration."Start-Stop"
	    THEN

	        #s_FB_MaintenanceCounter(ii_Group := #i_UDT_EquipmentNumber.Group,
	                                 ii_Node := #i_UDT_EquipmentNumber.Node,
	                                 idi_RunningTime := #sdi_RunningTime,
	                                 idi_DistanceTravelled := #sdi_DistanceTraveled,
	                                 "idi_Start-Stop" := #sdi_StartStop,
	                                 ii_MessageGroup := #ci_MessageGroup,
	                                 ix_FlagRetry := FALSE,
	                                 idi_TimeSpan := #ci_TimeSpan,
	                                 qx_Error => #sx_MaintenanceCounterBlockError,
	                                 qx_Warning => #sx_MaintenanceCounterBlockWarning,
	                                 iq_UDT_FifoHeader := #iq_UDT_FifoHeader,
	                                 iqs_FifoData := #iqs_FifoData,
	                                 iqdi_MessageSequenceNumber := #iqdi_MessageSequenceNumber);

	        #slr_RunningTimeMS := 0;
	        #sdi_RunningTime := 0;
	        #sdi_DistanceTraveled := 0;
	        #sdi_StartStop := 0;

	    END_IF;

	END_REGION

	REGION 8 - Write outputs

	    // Prepare collective output error.
	    #qx_Error :=
	    #sx_ItemErrorBlockError
	    OR #sx_ItemStatusBlockError
	    OR #sx_MaintenanceCounterBlockError
	    OR #sx_FIFOError;

	    // Prepare collective output warning.
	    #qx_Warning :=
	    #sx_ItemErrorBlockWarning
	    OR #sx_ItemStatusBlockWarning
	    OR #sx_MaintenanceCounterBlockWarning
	    OR #sx_FIFOWarning;

	END_REGION
END_FUNCTION_BLOCK

FUNCTION_BLOCK "FB_MFC_Visu_Caljan_Status"
{ S7_Optimized_Access := 'TRUE' }
VERSION : 2.0
// ATTRIBUTES
// AUTO_NUMBER = True
// BLOCK_NUMBER = 137
// END_ATTRIBUTES
   VAR_INPUT
      i_UDT_CaljanStatus { ExternalAccessible := 'False'; ExternalVisible := 'False'; ExternalWritable := 'False'} : "UDT_CaljanStatusV2";   // Caljan status structure
      i_UDT_EquipmentNumber { ExternalAccessible := 'False'; ExternalVisible := 'False'; ExternalWritable := 'False'} : "UDT_EquipmentNumber";   // Item number
      ix_SendAllErrorsState { ExternalAccessible := 'False'; ExternalVisible := 'False'; ExternalWritable := 'False'} : Bool;   // True - update all the messages
      ix_MFCConnected { ExternalAccessible := 'False'; ExternalVisible := 'False'; ExternalWritable := 'False'} : Bool;   // True - A connection to the MFC has been established
      ix_CollectiveReset { ExternalAccessible := 'False'; ExternalVisible := 'False'; ExternalWritable := 'False'} : Bool;   // True - Collective reset command of all system controls
   END_VAR

   VAR_OUTPUT
      qx_Error { ExternalAccessible := 'False'; ExternalVisible := 'False'; ExternalWritable := 'False'} : Bool;   // Block error
      qx_Warning { ExternalAccessible := 'False'; ExternalVisible := 'False'; ExternalWritable := 'False'} : Bool;   // Block warning
   END_VAR

   VAR_IN_OUT
      iq_UDT_FifoHeader : "UDT_FifoHeader";   // FIFO header
      iqs_FifoData : Array[*] of "UDT_MessageV2";   // FIFO data buffer
      iqdi_MessageSequenceNumber { ExternalAccessible := 'False'; ExternalVisible := 'False'; ExternalWritable := 'False'} : DInt;   // Message number
   END_VAR

   VAR
      s_FB_ItemError { ExternalAccessible := 'False'; ExternalVisible := 'False'; ExternalWritable := 'False'; S7_SetPoint := 'False'} : "FB_ItemError";   // Item error block's instance
      s_FB_ItemStatus { ExternalAccessible := 'False'; ExternalVisible := 'False'; ExternalWritable := 'False'; S7_SetPoint := 'False'} : "FB_ItemStatus";   // Item status block's instance
      ss_FIFOStatus { ExternalAccessible := 'False'; ExternalVisible := 'False'; ExternalWritable := 'False'; S7_SetPoint := 'False'} : "UDT_FifoStatus";   // Status structure
      s_UDT_Message { ExternalAccessible := 'False'; ExternalVisible := 'False'; ExternalWritable := 'False'; S7_SetPoint := 'False'} : "UDT_MessageV2";   // Message
      s_UDT_CaljanOld { ExternalAccessible := 'False'; ExternalVisible := 'False'; ExternalWritable := 'False'; S7_SetPoint := 'False'} : "UDT_CaljanStatusV2";   // Caljan status structure
      s_UDT_ItemError { ExternalAccessible := 'False'; ExternalVisible := 'False'; ExternalWritable := 'False'; S7_SetPoint := 'False'} : "UDT_ItemError";   // Item error message body structure
      s_UDT_ItemStatus { ExternalAccessible := 'False'; ExternalVisible := 'False'; ExternalWritable := 'False'; S7_SetPoint := 'False'} : "UDT_ItemStatus";   // Item status message body structure
      s_R_TRIG_Connection {InstructionName := 'R_TRIG'; LibVersion := '1.0'; ExternalAccessible := 'False'; ExternalVisible := 'False'; ExternalWritable := 'False'; S7_SetPoint := 'False'} : R_TRIG;   // Rising edge trigger connection reastablished
      s_F_TRIG_SendAllErrors {InstructionName := 'F_TRIG'; LibVersion := '1.0'; ExternalAccessible := 'False'; ExternalVisible := 'False'; ExternalWritable := 'False'; S7_SetPoint := 'False'} : F_TRIG;   // Falling edge trigger from signal send all errors
      sdi_Code { ExternalAccessible := 'False'; ExternalVisible := 'False'; ExternalWritable := 'False'} : DInt;   // Error code
      si_ItemStatus { ExternalAccessible := 'False'; ExternalVisible := 'False'; ExternalWritable := 'False'} : Int;   // Item status
      ii_ErrorNumber { ExternalAccessible := 'False'; ExternalVisible := 'False'; ExternalWritable := 'False'} : Int;   // Counter Error Number
      si_State { ExternalAccessible := 'False'; ExternalVisible := 'False'; ExternalWritable := 'False'} : Int;   // Error state
      sx_ItemErrorMessageReq { ExternalAccessible := 'False'; ExternalVisible := 'False'; ExternalWritable := 'False'} : Bool;   // Item error message required
      sx_ItemStatusMessageReq { ExternalAccessible := 'False'; ExternalVisible := 'False'; ExternalWritable := 'False'} : Bool;   // Item status message required
      sx_SendAllProcedure { ExternalAccessible := 'False'; ExternalVisible := 'False'; ExternalWritable := 'False'} : Bool;   // Send all procedure
      sx_FIFOError { ExternalAccessible := 'False'; ExternalVisible := 'False'; ExternalWritable := 'False'} : Bool;   // FIFO error
      sx_FIFOWarning { ExternalAccessible := 'False'; ExternalVisible := 'False'; ExternalWritable := 'False'} : Bool;   // FIFO warning
      sx_ItemErrorBlockError { ExternalAccessible := 'False'; ExternalVisible := 'False'; ExternalWritable := 'False'} : Bool;   // Item error block error
      sx_ItemErrorBlockWarning { ExternalAccessible := 'False'; ExternalVisible := 'False'; ExternalWritable := 'False'} : Bool;   // Item error block warning
      sx_ItemStatusBlockError { ExternalAccessible := 'False'; ExternalVisible := 'False'; ExternalWritable := 'False'} : Bool;   // Item status block error
      sx_ItemStatusBlockWarning { ExternalAccessible := 'False'; ExternalVisible := 'False'; ExternalWritable := 'False'} : Bool;   // Item status block warning
   END_VAR

   VAR_TEMP
      t_UDT_CaljanStatus : "UDT_CaljanStatusV2";   // Caljan status structure
   END_VAR


BEGIN
	(*
	----------------------------------------------------------------------------------------
	|                                                                                      |
	|  Copyright  2023             FORTNA Europe BV                                        |
	|  All Rights Reserved         Netherlands                                             |
	|                                                                                      |
	----------------------------------------------------------------------------------------
	Version history:
	Date        | Version   | Author       | Remark
	----------------------------------------------------------------------------------------
	21/03/2023  | 1.0       | M. Diebel   | Release TIA 17 | DHL Munich 2023
	05/09/2023  | 2.0       | M. Diebel   | Disable the information messages to MFC
	13/03/2023  | 2.1       | S. Nieswiec | Updated for new Baseline
	*)


	REGION 1 - Initialize message required signals

	    //Disable the information messages
	    // - Run mode
	    // - Store mode
	    // - Chute Disabled
	    // These information and statuses are generated in the Caljan conveyor but visuzalized in other elemenents of the 3D model
	    #t_UDT_CaljanStatus := #i_UDT_CaljanStatus;
	    #t_UDT_CaljanStatus.Specific.ChuteBlocked := FALSE;
	    #t_UDT_CaljanStatus.Specific.StoreMode := FALSE;
	    #t_UDT_CaljanStatus.Specific.RunMode := FALSE;

	    #sx_ItemErrorMessageReq := FALSE;
	    #sx_ItemStatusMessageReq := FALSE;

	    // On connection reestablish send last remembered status and error state ( status only when it's diffrent then 0 )
	    #s_R_TRIG_Connection(CLK := #ix_MFCConnected);

	    IF #s_R_TRIG_Connection.Q AND #si_ItemStatus <> 0
	    THEN
	        #sx_ItemStatusMessageReq := TRUE;
	    END_IF;

	    IF #s_R_TRIG_Connection.Q
	    THEN
	        #sx_ItemErrorMessageReq := TRUE;
	    END_IF;

	    // Prepare trigger on the collective reset signal.
	    #s_F_TRIG_SendAllErrors(CLK := #ix_SendAllErrorsState);

	    // When collective reset will go down, start send every equipment errors.
	    IF #s_F_TRIG_SendAllErrors.Q AND NOT #sx_SendAllProcedure
	    THEN
	        #ii_ErrorNumber := 0;
	        #sx_SendAllProcedure := TRUE;
	    END_IF;

	END_REGION

	REGION 2 - FIFO header status update

	    // Mode 'S' - FIFO register status update.
	    "FC_Fifo"(ic_Mode := 'S',
	              qUDT_Status => #ss_FIFOStatus,
	              qx_Error => #sx_FIFOError,
	              qx_Warning => #sx_FIFOWarning,
	              iqv_Data := #s_UDT_Message,
	              iqUDT_FifoHeader := #iq_UDT_FifoHeader,
	              iqv_DataBuffer := #iqs_FifoData);

	END_REGION

	REGION 3 - Prepare message data

	    // When there is no reset errors command, update status and errors.
	    IF NOT #ix_CollectiveReset
	        AND NOT #ss_FIFOStatus.FifoPreFull
	    THEN
	        // Status
	        IF (#t_UDT_CaljanStatus.Status <> #s_UDT_CaljanOld.Status OR (#sx_SendAllProcedure AND #ii_ErrorNumber = 0))
	        THEN
	            #sx_ItemStatusMessageReq := TRUE;
	            #si_ItemStatus := #t_UDT_CaljanStatus.Status;
	            #s_UDT_CaljanOld.Status := #t_UDT_CaljanStatus.Status;
	        END_IF;


	        // Check which specific status changed, prepare code, change state and write new status into the old one.
	        IF (#t_UDT_CaljanStatus.Specific.PNSlaveNotOnline <> #s_UDT_CaljanOld.Specific.PNSlaveNotOnline AND NOT #sx_SendAllProcedure)
	            OR (#sx_SendAllProcedure AND #ii_ErrorNumber = 0)
	        THEN
	            #sdi_Code := "DB_MFC_ErrorCode".Caljan.PNSlaveNotOnline;
	            #si_State := BOOL_TO_INT(#t_UDT_CaljanStatus.Specific.PNSlaveNotOnline);
	            #s_UDT_CaljanOld.Specific.PNSlaveNotOnline := #t_UDT_CaljanStatus.Specific.PNSlaveNotOnline;
	            #sx_ItemErrorMessageReq := TRUE;
	            #ii_ErrorNumber += 1;
	        ELSIF (#t_UDT_CaljanStatus.Specific.PNSlaveError <> #s_UDT_CaljanOld.Specific.PNSlaveError AND NOT #sx_SendAllProcedure)
	            OR (#sx_SendAllProcedure AND #ii_ErrorNumber = 1)
	        THEN
	            #sdi_Code := "DB_MFC_ErrorCode".Caljan.PNSlaveError;
	            #si_State := BOOL_TO_INT(#t_UDT_CaljanStatus.Specific.PNSlaveError);
	            #s_UDT_CaljanOld.Specific.PNSlaveError := #t_UDT_CaljanStatus.Specific.PNSlaveError;
	            #sx_ItemErrorMessageReq := TRUE;
	            #ii_ErrorNumber += 1;
	        ELSIF (#t_UDT_CaljanStatus.Specific.PNSlaveWarning <> #s_UDT_CaljanOld.Specific.PNSlaveWarning AND NOT #sx_SendAllProcedure)
	            OR (#sx_SendAllProcedure AND #ii_ErrorNumber = 2)
	        THEN
	            #sdi_Code := "DB_MFC_ErrorCode".Caljan.PNSlaveWarning;
	            #si_State := BOOL_TO_INT(#t_UDT_CaljanStatus.Specific.PNSlaveWarning);
	            #s_UDT_CaljanOld.Specific.PNSlaveWarning := #t_UDT_CaljanStatus.Specific.PNSlaveWarning;
	            #sx_ItemErrorMessageReq := TRUE;
	            #ii_ErrorNumber += 1;
	        ELSIF (#t_UDT_CaljanStatus.Specific.Disabled <> #s_UDT_CaljanOld.Specific.Disabled AND NOT #sx_SendAllProcedure)
	            OR (#sx_SendAllProcedure AND #ii_ErrorNumber = 3)
	        THEN
	            #sdi_Code := "DB_MFC_ErrorCode".Caljan.Disabled;
	            #si_State := BOOL_TO_INT(#t_UDT_CaljanStatus.Specific.Disabled);
	            #s_UDT_CaljanOld.Specific.Disabled := #t_UDT_CaljanStatus.Specific.Disabled;
	            #sx_ItemErrorMessageReq := TRUE;
	            #ii_ErrorNumber += 1;
	        ELSIF (#t_UDT_CaljanStatus.Specific.VFDError <> #s_UDT_CaljanOld.Specific.VFDError AND NOT #sx_SendAllProcedure)
	            OR (#sx_SendAllProcedure AND #ii_ErrorNumber = 4)
	        THEN
	            #sdi_Code := "DB_MFC_ErrorCode".Caljan.VFDError;
	            #si_State := BOOL_TO_INT(#t_UDT_CaljanStatus.Specific.VFDError);
	            #s_UDT_CaljanOld.Specific.VFDError := #t_UDT_CaljanStatus.Specific.VFDError;
	            #sx_ItemErrorMessageReq := TRUE;
	            #ii_ErrorNumber += 1;
	        ELSIF (#t_UDT_CaljanStatus.Specific.NotHealthy <> #s_UDT_CaljanOld.Specific.NotHealthy AND NOT #sx_SendAllProcedure)
	            OR (#sx_SendAllProcedure AND #ii_ErrorNumber = 5)
	        THEN
	            #sdi_Code := "DB_MFC_ErrorCode".Caljan.NotHealthy;
	            #si_State := BOOL_TO_INT(#t_UDT_CaljanStatus.Specific.NotHealthy);
	            #s_UDT_CaljanOld.Specific.NotHealthy := #t_UDT_CaljanStatus.Specific.NotHealthy;
	            #sx_ItemErrorMessageReq := TRUE;
	            #ii_ErrorNumber += 1;
	        ELSIF (#t_UDT_CaljanStatus.Specific.StoreMode <> #s_UDT_CaljanOld.Specific.StoreMode AND NOT #sx_SendAllProcedure)
	            OR (#sx_SendAllProcedure AND #ii_ErrorNumber = 6)
	        THEN
	            #sdi_Code := "DB_MFC_ErrorCode".Caljan.StoreMode;
	            #si_State := BOOL_TO_INT(#t_UDT_CaljanStatus.Specific.StoreMode);
	            #s_UDT_CaljanOld.Specific.StoreMode := #t_UDT_CaljanStatus.Specific.StoreMode;
	            #sx_ItemErrorMessageReq := TRUE;
	            #ii_ErrorNumber += 1;
	        ELSIF (#t_UDT_CaljanStatus.Specific.RunMode <> #s_UDT_CaljanOld.Specific.RunMode AND NOT #sx_SendAllProcedure)
	            OR (#sx_SendAllProcedure AND #ii_ErrorNumber = 7)
	        THEN
	            #sdi_Code := "DB_MFC_ErrorCode".Caljan.RunMode;
	            #si_State := BOOL_TO_INT(#t_UDT_CaljanStatus.Specific.RunMode);
	            #s_UDT_CaljanOld.Specific.RunMode := #t_UDT_CaljanStatus.Specific.RunMode;
	            #sx_ItemErrorMessageReq := TRUE;
	            #ii_ErrorNumber += 1;
	        ELSIF (#t_UDT_CaljanStatus.Specific.ChuteBlocked <> #s_UDT_CaljanOld.Specific.ChuteBlocked AND NOT #sx_SendAllProcedure)
	            OR (#sx_SendAllProcedure AND #ii_ErrorNumber = 8)
	        THEN
	            #sdi_Code := "DB_MFC_ErrorCode".Caljan.ChuteBlocked;
	            #si_State := BOOL_TO_INT(#t_UDT_CaljanStatus.Specific.ChuteBlocked);
	            #s_UDT_CaljanOld.Specific.ChuteBlocked := #t_UDT_CaljanStatus.Specific.ChuteBlocked;
	            #sx_ItemErrorMessageReq := TRUE;
	            #ii_ErrorNumber += 1;

	        ELSIF (#t_UDT_CaljanStatus.Specific.PEC_EoS.PEC <> #s_UDT_CaljanOld.Specific.PEC_EoS.PEC AND NOT #sx_SendAllProcedure)
	            OR (#sx_SendAllProcedure AND #ii_ErrorNumber = 9)
	        THEN
	            #sx_ItemErrorMessageReq := TRUE;
	            #s_UDT_CaljanOld.Specific.PEC_EoS.PEC := #t_UDT_CaljanStatus.Specific.PEC_EoS.PEC;
	            #ii_ErrorNumber += 1;
	        ELSIF (#t_UDT_CaljanStatus.Specific.PEC_EoS.Jam <> #s_UDT_CaljanOld.Specific.PEC_EoS.Jam AND NOT #sx_SendAllProcedure)
	            OR (#sx_SendAllProcedure AND #ii_ErrorNumber = 10)
	        THEN
	            #sdi_Code := "DB_MFC_ErrorCode".Caljan.Jam;
	            #si_State := BOOL_TO_INT(#t_UDT_CaljanStatus.Specific.PEC_EoS.Jam);
	            #s_UDT_CaljanOld.Specific.PEC_EoS.Jam := #t_UDT_CaljanStatus.Specific.PEC_EoS.Jam;
	            #sx_ItemErrorMessageReq := TRUE;
	            #sx_SendAllProcedure := FALSE;
	        END_IF;
	    END_IF;
	END_REGION

	REGION 4 - Write message components to the item error structure

	    #s_UDT_ItemError.ItemNumber := #i_UDT_EquipmentNumber;
	    #s_UDT_ItemError.Error := #sdi_Code;
	    #s_UDT_ItemError.State := #si_State;
	    #s_UDT_ItemError.Masked := 1;

	END_REGION

	REGION 5 - Write message components to the item status structure

	    #s_UDT_ItemStatus.Group := #i_UDT_EquipmentNumber.Group;
	    #s_UDT_ItemStatus.Node := #i_UDT_EquipmentNumber.Node;
	    #s_UDT_ItemStatus.Status := #si_ItemStatus;

	END_REGION

	REGION 6 - Prepare messages to the MFC

	    // If item error message required signal is set, prepare the item error message.
	    IF (#sx_ItemErrorMessageReq)
	    THEN
	        #s_FB_ItemError(i_UDT_ItemErrorBody := #s_UDT_ItemError,
	                        ii_MessageGroup := 1,
	                        ix_FlagRetry := FALSE,
	                        idi_TimeSpan := 0,
	                        qx_Error => #sx_ItemErrorBlockError,
	                        qx_Warning => #sx_ItemErrorBlockWarning,
	                        iq_UDT_FifoHeader := #iq_UDT_FifoHeader,
	                        iqs_FifoData := #iqs_FifoData,
	                        iqdi_MessageSequenceNumber := #iqdi_MessageSequenceNumber);
	    END_IF;

	    // If item status message required signal is set, prepare the item error message.
	    IF (#sx_ItemStatusMessageReq)
	    THEN
	        #s_FB_ItemStatus(i_UDT_ItemStatusBody := #s_UDT_ItemStatus,
	                         ii_MessageGroup := 1,
	                         ix_FlagRetry := FALSE,
	                         idi_TimeSpan := 0,
	                         qx_Error => #sx_ItemStatusBlockError,
	                         qx_Warning => #sx_ItemStatusBlockWarning,
	                         iq_UDT_FifoHeader := #iq_UDT_FifoHeader,
	                         iqs_FifoData := #iqs_FifoData,
	                         iqdi_MessageSequenceNumber := #iqdi_MessageSequenceNumber);
	    END_IF;

	END_REGION

	REGION 7 - Write outputs

	    // Prepare collective output error.
	    #qx_Error :=
	    #sx_ItemErrorBlockError
	    OR #sx_ItemStatusBlockError
	    OR #sx_FIFOError;

	    // Prepare collective output warning.
	    #qx_Warning :=
	    #sx_ItemErrorBlockWarning
	    OR #sx_ItemStatusBlockWarning
	    OR #sx_FIFOWarning;

	END_REGION





END_FUNCTION_BLOCK

FUNCTION_BLOCK "FB_MFC_Visu_VFD_Status"
{ S7_Optimized_Access := 'TRUE' }
VERSION : 0.1
// ATTRIBUTES
// AUTO_NUMBER = True
// BLOCK_NUMBER = 163
// END_ATTRIBUTES
   VAR_INPUT
      ix_SendAllErrorsState { ExternalAccessible := 'False'; ExternalVisible := 'False'; ExternalWritable := 'False'} : Bool;   // True - update all the messages
      ix_MFCConnected { ExternalAccessible := 'False'; ExternalVisible := 'False'; ExternalWritable := 'False'} : Bool;   // True - A connection to the MFC has been established
      ix_CollectiveReset { ExternalAccessible := 'False'; ExternalVisible := 'False'; ExternalWritable := 'False'} : Bool;   // True - Collective reset command of all system controls
      iUDT_VFDStatus { ExternalAccessible := 'False'; ExternalVisible := 'False'; ExternalWritable := 'False'} : "UDT_VfdStatus";   // VFD status structrue
      iUDT_EquipmentNumber { ExternalAccessible := 'False'; ExternalVisible := 'False'; ExternalWritable := 'False'} : "UDT_EquipmentNumber";   // Equipment Number
   END_VAR

   VAR_OUTPUT
      qx_Error { ExternalAccessible := 'False'; ExternalVisible := 'False'; ExternalWritable := 'False'} : Bool;   // Block error
      qx_Warning { ExternalAccessible := 'False'; ExternalVisible := 'False'; ExternalWritable := 'False'} : Bool;   // Block warning
   END_VAR

   VAR_IN_OUT
      iqUDT_FifoHeader : "UDT_FifoHeader";   // FIFO header
      iqsFifoData : Array[*] of "UDT_MessageV2";   // FIFO data buffer
      iqdi_MessageSequenceNumber { ExternalAccessible := 'False'; ExternalVisible := 'False'; ExternalWritable := 'False'} : DInt;   // Message number
   END_VAR

   VAR
      s_FB_ItemError { ExternalAccessible := 'False'; ExternalVisible := 'False'; ExternalWritable := 'False'; S7_SetPoint := 'False'} : "FB_ItemError";   // Item error block's instance
      s_UDT_Message { ExternalAccessible := 'False'; ExternalVisible := 'False'; ExternalWritable := 'False'; S7_SetPoint := 'False'} : "UDT_BytesMessage";   // Message
      s_UDT_ItemError { ExternalAccessible := 'False'; ExternalVisible := 'False'; ExternalWritable := 'False'; S7_SetPoint := 'False'} : "UDT_ItemError";   // Item error message body structure
      "i_UDT_VFDStatus.OLD" { ExternalAccessible := 'False'; ExternalVisible := 'False'; ExternalWritable := 'False'; S7_SetPoint := 'False'} : "UDT_VfdStatus";   // VFD old status structure
      ss_FIFOStatus { ExternalAccessible := 'False'; ExternalVisible := 'False'; ExternalWritable := 'False'; S7_SetPoint := 'False'} : "UDT_FifoStatus";   // Status structure
      s_R_TRIG_Connection {InstructionName := 'R_TRIG'; LibVersion := '1.0'; ExternalAccessible := 'False'; ExternalVisible := 'False'; ExternalWritable := 'False'; S7_SetPoint := 'False'} : R_TRIG;   // Rising edge trigger connection reastablished
      s_F_TRIG_SendAllErrors {InstructionName := 'F_TRIG'; LibVersion := '1.0'; ExternalAccessible := 'False'; ExternalVisible := 'False'; ExternalWritable := 'False'; S7_SetPoint := 'False'} : F_TRIG;   // Falling edge trigger from signal send all errors
      sdi_Code { ExternalAccessible := 'False'; ExternalVisible := 'False'; ExternalWritable := 'False'} : DInt;   // Error code
      si_State { ExternalAccessible := 'False'; ExternalVisible := 'False'; ExternalWritable := 'False'} : Int;   // Error state
      ii_ErrorNumber { ExternalAccessible := 'False'; ExternalVisible := 'False'; ExternalWritable := 'False'} : Int;   // Counter "Error Number"
      sx_ItemErrorMessageReq { ExternalAccessible := 'False'; ExternalVisible := 'False'; ExternalWritable := 'False'} : Bool;   // Item error message required
      sx_ItemErrorBlockError { ExternalAccessible := 'False'; ExternalVisible := 'False'; ExternalWritable := 'False'} : Bool;   // Item error block error
      sx_ItemErrorBlockWarning { ExternalAccessible := 'False'; ExternalVisible := 'False'; ExternalWritable := 'False'} : Bool;   // Item error block warning
      sx_SendAllProcedure { ExternalAccessible := 'False'; ExternalVisible := 'False'; ExternalWritable := 'False'} : Bool;   // Send all procedure
      sx_FIFOError { ExternalAccessible := 'False'; ExternalVisible := 'False'; ExternalWritable := 'False'} : Bool;   // FIFO Error
      sx_FIFOWarning { ExternalAccessible := 'False'; ExternalVisible := 'False'; ExternalWritable := 'False'} : Bool;   // FIFO Warning
      sx_FirstCycle { ExternalAccessible := 'False'; ExternalVisible := 'False'; ExternalWritable := 'False'} : Bool;
   END_VAR


BEGIN
	(*
	----------------------------------------------------------------------------------------
	|                                                                                      |
	|  Copyright  2023             FORTNA Europe BV                                        |
	|  All Rights Reserved         Netherlands                                             |
	|                                                                                      |
	----------------------------------------------------------------------------------------
	Version history:
	Date        | Version   | Author       | Remark
	----------------------------------------------------------------------------------------
	03/01/2023  | 1.0       | S. Nikodem   | Release TIA 17     | DHL Munich 2023
	11/08/2023  | 1.1       | M.Diebel     | Send all procedure | DHL Munich 2023
	13/03/2023  | 1.2       | S. Nieswiec  | Updated for new Baseline
	*)

	REGION 1 - Initialize message required signals

	    #sx_ItemErrorMessageReq := FALSE;

	    // On connection reestablish send last remembered status and error state ( status only when it's diffrent then 0 )
	    #s_R_TRIG_Connection(CLK := #ix_MFCConnected);


	    IF #s_R_TRIG_Connection.Q
	    THEN
	        #sx_SendAllProcedure := TRUE;
	        #ii_ErrorNumber := 0;
	    END_IF;

	    // Prepare trigger on the collective reset signal.
	    #s_F_TRIG_SendAllErrors(CLK := #ix_SendAllErrorsState);

	    // When collective reset will go down, start send every equipment errors.
	    IF #s_F_TRIG_SendAllErrors.Q AND NOT #sx_SendAllProcedure
	    THEN
	        #ii_ErrorNumber := 0;
	        #sx_SendAllProcedure := TRUE;
	    END_IF;

	END_REGION

	REGION 2 - FIFO header status update

	    // Mode 'S' - FIFO register status update.
	    "FC_Fifo"(ic_Mode := 'S',
	              qUDT_Status => #ss_FIFOStatus,
	              qx_Error => #sx_FIFOError,
	              qx_Warning => #sx_FIFOWarning,
	              iqv_Data := #s_UDT_Message,
	              iqUDT_FifoHeader := #iqUDT_FifoHeader,
	              iqv_DataBuffer := #iqsFifoData);

	END_REGION

	REGION 3 - Prepare message data

	    // When there is no reset errors command, update status and errors.
	    IF NOT #ix_CollectiveReset
	        AND NOT #ss_FIFOStatus.FifoPreFull
	    THEN


	        // If the status changed, set item error message required signal.
	        IF (#iUDT_VFDStatus <> #"i_UDT_VFDStatus.OLD" OR #sx_SendAllProcedure OR #sx_FirstCycle)
	        THEN
	            #sx_ItemErrorMessageReq := TRUE;

	            #"i_UDT_VFDStatus.OLD".ErrorCode := #iUDT_VFDStatus.ErrorCode;
	            #"i_UDT_VFDStatus.OLD".SubErrorCode := #iUDT_VFDStatus.SubErrorCode;

	            // Check which specific status changed, prepare code, change state and write new status into the old one.
	            IF (#iUDT_VFDStatus.CommunicationErrorMovikit <> #"i_UDT_VFDStatus.OLD".CommunicationErrorMovikit AND NOT #sx_SendAllProcedure)
	                OR ((#sx_SendAllProcedure OR #sx_FirstCycle) AND #ii_ErrorNumber = 0)
	            THEN
	                #sdi_Code := "DB_MFC_ErrorCode".VFD.CommunicationErrorMovikit;
	                #si_State := BOOL_TO_INT(#iUDT_VFDStatus.CommunicationErrorMovikit);
	                #"i_UDT_VFDStatus.OLD".CommunicationErrorMovikit := #iUDT_VFDStatus.CommunicationErrorMovikit;
	                #ii_ErrorNumber += 1;
	            ELSIF (#iUDT_VFDStatus.InternalError <> #"i_UDT_VFDStatus.OLD".InternalError AND NOT #sx_SendAllProcedure)
	                OR ((#sx_SendAllProcedure OR #sx_FirstCycle) AND #ii_ErrorNumber = 1)
	            THEN
	                #sdi_Code := "DB_MFC_ErrorCode".VFD.InternalError;
	                #si_State := BOOL_TO_INT(#iUDT_VFDStatus.InternalError);
	                #"i_UDT_VFDStatus.OLD".InternalError := #iUDT_VFDStatus.InternalError;
	                #ii_ErrorNumber += 1;
	            ELSIF (#iUDT_VFDStatus.InternalWarning <> #"i_UDT_VFDStatus.OLD".InternalWarning AND NOT #sx_SendAllProcedure)
	                OR ((#sx_SendAllProcedure OR #sx_FirstCycle) AND #ii_ErrorNumber = 2)
	            THEN
	                #sdi_Code := "DB_MFC_ErrorCode".VFD.InternalWarning;
	                #si_State := BOOL_TO_INT(#iUDT_VFDStatus.InternalWarning);
	                #"i_UDT_VFDStatus.OLD".InternalWarning := #iUDT_VFDStatus.InternalWarning;
	                #ii_ErrorNumber += 1;
	                // ELSIF (#i_UDT_VFDStatus.OutOfPosition_Error <> #i_UDT_VFDStatus.OLD.OutOfPosition_Error AND NOT #sx_SendAllProcedure)
	                //     OR (#sx_SendAllProcedure AND #ii_ErrorNumber = 3)
	                // THEN
	                //     #sdi_Code := 104;
	                //     #si_State := BOOL_TO_INT(#i_UDT_VFDStatus..OutOfPosition_Error);
	                //     #i_UDT_VFDStatus.OLD.OutOfPosition_Error := #i_UDT_VFDStatus.OutOfPosition_Error;
	                //     #ii_ErrorNumber += 1;
	            ELSIF (#iUDT_VFDStatus.PNSlaveError <> #"i_UDT_VFDStatus.OLD".PNSlaveError AND NOT #sx_SendAllProcedure)
	                OR ((#sx_SendAllProcedure OR #sx_FirstCycle) AND #ii_ErrorNumber = 3)
	            THEN
	                #sdi_Code := "DB_MFC_ErrorCode".VFD.PNSlaveError;
	                #si_State := BOOL_TO_INT(#iUDT_VFDStatus.PNSlaveError);
	                #"i_UDT_VFDStatus.OLD".PNSlaveError := #iUDT_VFDStatus.PNSlaveError;
	                #ii_ErrorNumber += 1;
	            ELSIF (#iUDT_VFDStatus.PNSlaveNotonline <> #"i_UDT_VFDStatus.OLD".PNSlaveNotonline AND NOT #sx_SendAllProcedure)
	                OR ((#sx_SendAllProcedure OR #sx_FirstCycle) AND #ii_ErrorNumber = 4)
	            THEN
	                #sdi_Code := "DB_MFC_ErrorCode".VFD.PNSlaveNotonline;
	                #si_State := BOOL_TO_INT(#iUDT_VFDStatus.PNSlaveNotonline);
	                #"i_UDT_VFDStatus.OLD".PNSlaveNotonline := #iUDT_VFDStatus.PNSlaveNotonline;
	                #ii_ErrorNumber += 1;
	            ELSIF (#iUDT_VFDStatus.PNSlaveWarning <> #"i_UDT_VFDStatus.OLD".PNSlaveWarning AND NOT #sx_SendAllProcedure)
	                OR ((#sx_SendAllProcedure OR #sx_FirstCycle) AND #ii_ErrorNumber = 5)
	            THEN
	                #sdi_Code := "DB_MFC_ErrorCode".VFD.PNSlaveWarning;
	                #si_State := BOOL_TO_INT(#iUDT_VFDStatus.PNSlaveWarning);
	                #"i_UDT_VFDStatus.OLD".PNSlaveWarning := #iUDT_VFDStatus.PNSlaveWarning;
	                #ii_ErrorNumber += 1;
	            ELSIF (#iUDT_VFDStatus.VFDRunningFeedbackError <> #"i_UDT_VFDStatus.OLD".VFDRunningFeedbackError AND NOT #sx_SendAllProcedure)
	                OR ((#sx_SendAllProcedure OR #sx_FirstCycle) AND #ii_ErrorNumber = 6)
	            THEN
	                #sdi_Code := "DB_MFC_ErrorCode".VFD.VFDRunningFeedbackError;
	                #si_State := BOOL_TO_INT(#iUDT_VFDStatus.VFDRunningFeedbackError);
	                #"i_UDT_VFDStatus.OLD".VFDRunningFeedbackError := #iUDT_VFDStatus.VFDRunningFeedbackError;
	                #sx_SendAllProcedure := FALSE;
	                #sx_FirstCycle := FALSE;
	            END_IF;

	            // // Prepare the alarm word.
	            // #qw_AlarmWord1.%X0 := #i_UDT_VFDStatus..CommunicationErrorMovikit;
	            // #qw_AlarmWord1.%X1 := #i_UDT_VFDStatus..InternalError;
	            // #qw_AlarmWord1.%X2 := #i_UDT_VFDStatus..InternalWarning;
	            // #qw_AlarmWord1.%X3 := #i_UDT_VFDStatus..OutOfPosition_Error;
	            // #qw_AlarmWord1.%X4 := #i_UDT_VFDStatus..PNSlaveError;
	            // #qw_AlarmWord1.%X5 := #i_UDT_VFDStatus..PNSlaveNotonline;
	            // #qw_AlarmWord1.%X6 := #i_UDT_VFDStatus..PNSlaveWarning;

	        END_IF;

	    END_IF;

	END_REGION

	REGION 4 - Write message components to the item error structure

	    #s_UDT_ItemError.ItemNumber := #iUDT_EquipmentNumber;
	    #s_UDT_ItemError.Error := #sdi_Code;
	    #s_UDT_ItemError.State := #si_State;
	    #s_UDT_ItemError.Masked := 1;

	END_REGION

	REGION 5 - Prepare messages to the MFC

	    // If item error message required signal is set, prepare the item error message.
	    IF (#sx_ItemErrorMessageReq)
	    THEN
	        #s_FB_ItemError(i_UDT_ItemErrorBody := #s_UDT_ItemError,
	                        ii_MessageGroup := 1,
	                        ix_FlagRetry := FALSE,
	                        idi_TimeSpan := 0,
	                        qx_Error => #sx_ItemErrorBlockError,
	                        qx_Warning => #sx_ItemErrorBlockWarning,
	                        iq_UDT_FifoHeader := #iqUDT_FifoHeader,
	                        iqs_FifoData := #iqsFifoData,
	                        iqdi_MessageSequenceNumber := #iqdi_MessageSequenceNumber);
	    END_IF;

	END_REGION

	REGION 6 - Write outputs

	    // Prepare collective output error.
	    #qx_Error := #sx_ItemErrorBlockError
	    OR #sx_FIFOError;

	    // Prepare collective output warning.
	    #qx_Warning := #sx_ItemErrorBlockWarning
	    OR #sx_FIFOWarning;

	END_REGION
END_FUNCTION_BLOCK

FUNCTION_BLOCK "FB_MFC_Visu_ColumnLift_Status"
{ S7_Optimized_Access := 'TRUE' }
VERSION : 2.0
// ATTRIBUTES
// AUTO_NUMBER = True
// BLOCK_NUMBER = 139
// END_ATTRIBUTES
   VAR_INPUT
      i_UDT_ColumnLiftStatus { ExternalAccessible := 'False'; ExternalVisible := 'False'; ExternalWritable := 'False'} : "UDT_ColumnLift_Status";
      i_UDT_EquipmentNumber { ExternalAccessible := 'False'; ExternalVisible := 'False'; ExternalWritable := 'False'} : "UDT_EquipmentNumber";   // Item number
      ix_SendAllErrorsState { ExternalAccessible := 'False'; ExternalVisible := 'False'; ExternalWritable := 'False'} : Bool;   // True - update all the messages
      ix_MFCConnected { ExternalAccessible := 'False'; ExternalVisible := 'False'; ExternalWritable := 'False'} : Bool;   // True - A connection to the MFC has been established
      ix_CollectiveReset { ExternalAccessible := 'False'; ExternalVisible := 'False'; ExternalWritable := 'False'} : Bool;   // True - Collective reset command of all system controls
   END_VAR

   VAR_OUTPUT
      qx_Error { ExternalAccessible := 'False'; ExternalVisible := 'False'; ExternalWritable := 'False'} : Bool;   // Block error
      qx_Warning { ExternalAccessible := 'False'; ExternalVisible := 'False'; ExternalWritable := 'False'} : Bool;   // Block warning
   END_VAR

   VAR_IN_OUT
      iq_UDT_FifoHeader : "UDT_FifoHeader";   // FIFO header
      iqs_FifoData : Array[*] of "UDT_MessageV2";   // FIFO data buffer
      iqdi_MessageSequenceNumber { ExternalAccessible := 'False'; ExternalVisible := 'False'; ExternalWritable := 'False'} : DInt;   // Message number
   END_VAR

   VAR
      s_FB_ItemError { ExternalAccessible := 'False'; ExternalVisible := 'False'; ExternalWritable := 'False'; S7_SetPoint := 'False'} : "FB_ItemError";   // Item error block's instance
      s_FB_ItemStatus { ExternalAccessible := 'False'; ExternalVisible := 'False'; ExternalWritable := 'False'; S7_SetPoint := 'False'} : "FB_ItemStatus";   // Item status block's instance
      ss_FIFOStatus { ExternalAccessible := 'False'; ExternalVisible := 'False'; ExternalWritable := 'False'; S7_SetPoint := 'False'} : "UDT_FifoStatus";   // Status structure
      s_UDT_Message { ExternalAccessible := 'False'; ExternalVisible := 'False'; ExternalWritable := 'False'; S7_SetPoint := 'False'} : "UDT_MessageV2";   // Message
      s_UDT_ColumnLiftOld { ExternalAccessible := 'False'; ExternalVisible := 'False'; ExternalWritable := 'False'; S7_SetPoint := 'False'} : "UDT_ColumnLift_Status";   // ColumnLift status structure
      s_UDT_ItemError { ExternalAccessible := 'False'; ExternalVisible := 'False'; ExternalWritable := 'False'; S7_SetPoint := 'False'} : "UDT_ItemError";   // Item error message body structure
      s_UDT_ItemStatus { ExternalAccessible := 'False'; ExternalVisible := 'False'; ExternalWritable := 'False'; S7_SetPoint := 'False'} : "UDT_ItemStatus";   // Item status message body structure
      s_R_TRIG_Connection {InstructionName := 'R_TRIG'; LibVersion := '1.0'; ExternalAccessible := 'False'; ExternalVisible := 'False'; ExternalWritable := 'False'; S7_SetPoint := 'False'} : R_TRIG;   // Rising edge trigger connection reastablished
      s_F_TRIG_SendAllErrors {InstructionName := 'F_TRIG'; LibVersion := '1.0'; ExternalAccessible := 'False'; ExternalVisible := 'False'; ExternalWritable := 'False'; S7_SetPoint := 'False'} : F_TRIG;   // Falling edge trigger from signal send all errors
      sdi_Code { ExternalAccessible := 'False'; ExternalVisible := 'False'; ExternalWritable := 'False'} : DInt;   // Error code
      si_ItemStatus { ExternalAccessible := 'False'; ExternalVisible := 'False'; ExternalWritable := 'False'} : Int;   // Item status
      ii_ErrorNumber { ExternalAccessible := 'False'; ExternalVisible := 'False'; ExternalWritable := 'False'} : Int;   // Counter Error Number
      si_State { ExternalAccessible := 'False'; ExternalVisible := 'False'; ExternalWritable := 'False'} : Int;   // Error state
      sx_ItemErrorMessageReq { ExternalAccessible := 'False'; ExternalVisible := 'False'; ExternalWritable := 'False'} : Bool;   // Item error message required
      sx_ItemStatusMessageReq { ExternalAccessible := 'False'; ExternalVisible := 'False'; ExternalWritable := 'False'} : Bool;   // Item status message required
      sx_SendAllProcedure { ExternalAccessible := 'False'; ExternalVisible := 'False'; ExternalWritable := 'False'} : Bool;   // Send all procedure
      sx_FIFOError { ExternalAccessible := 'False'; ExternalVisible := 'False'; ExternalWritable := 'False'} : Bool;   // FIFO error
      sx_FIFOWarning { ExternalAccessible := 'False'; ExternalVisible := 'False'; ExternalWritable := 'False'} : Bool;   // FIFO warning
      sx_ItemErrorBlockError { ExternalAccessible := 'False'; ExternalVisible := 'False'; ExternalWritable := 'False'} : Bool;   // Item error block error
      sx_ItemErrorBlockWarning { ExternalAccessible := 'False'; ExternalVisible := 'False'; ExternalWritable := 'False'} : Bool;   // Item error block warning
      sx_ItemStatusBlockError { ExternalAccessible := 'False'; ExternalVisible := 'False'; ExternalWritable := 'False'} : Bool;   // Item status block error
      sx_ItemStatusBlockWarning { ExternalAccessible := 'False'; ExternalVisible := 'False'; ExternalWritable := 'False'} : Bool;   // Item status block warning
   END_VAR

   VAR_TEMP
      t_UDT_ColumnLiftStatus : "UDT_ColumnLift_Status";   // ColumnLift status structure
   END_VAR


BEGIN
	(*
	----------------------------------------------------------------------------------------
	|                                                                                      |
	|  Copyright  2023             FORTNA Europe BV                                        |
	|  All Rights Reserved         Netherlands                                             |
	|                                                                                      |
	----------------------------------------------------------------------------------------
	Version history:
	Date        | Version   | Author       | Remark
	----------------------------------------------------------------------------------------
	24/04/2023  | 1.0       | M. Diebel   | Release TIA 17 | DHL Munich 2023
	11/09/2023  | 2.0       | M. Diebel   | Disable the information messages to MFC
	13/03/2023  | 2.1       | S. Nieswiec  | Updated for new Baseline
	*)


	REGION 1 - Initialize message required signals
	    //Move input to temp
	    #t_UDT_ColumnLiftStatus := #i_UDT_ColumnLiftStatus;
	    //Disable the information messages
	    //-UpperPosition
	    //-LowerPosition
	    #t_UDT_ColumnLiftStatus.Specific.UpperPosition := False;
	    #t_UDT_ColumnLiftStatus.Specific.LowerPosition := False;


	    #sx_ItemErrorMessageReq := FALSE;
	    #sx_ItemStatusMessageReq := FALSE;

	    // On connection reestablish send last remembered status and error state ( status only when it's diffrent then 0 )
	    #s_R_TRIG_Connection(CLK := #ix_MFCConnected);

	    IF #s_R_TRIG_Connection.Q AND #si_ItemStatus <> 0
	    THEN
	        #sx_ItemStatusMessageReq := TRUE;
	    END_IF;

	    IF #s_R_TRIG_Connection.Q
	    THEN
	        #sx_ItemErrorMessageReq := TRUE;
	    END_IF;

	    // Prepare trigger on the collective reset signal.
	    #s_F_TRIG_SendAllErrors(CLK := #ix_SendAllErrorsState);

	    // When collective reset will go down, start send every equipment errors.
	    IF #s_F_TRIG_SendAllErrors.Q AND NOT #sx_SendAllProcedure
	    THEN
	        #ii_ErrorNumber := 0;
	        #sx_SendAllProcedure := TRUE;
	    END_IF;

	END_REGION

	REGION 2 - FIFO header status update

	    // Mode 'S' - FIFO register status update.
	    "FC_Fifo"(ic_Mode := 'S',
	              qUDT_Status => #ss_FIFOStatus,
	              qx_Error => #sx_FIFOError,
	              qx_Warning => #sx_FIFOWarning,
	              iqv_Data := #s_UDT_Message,
	              iqUDT_FifoHeader := #iq_UDT_FifoHeader,
	              iqv_DataBuffer := #iqs_FifoData);

	END_REGION

	REGION 3 - Prepare message data

	    // When there is no reset errors command, update status and errors.
	    IF NOT #ix_CollectiveReset
	        AND NOT #ss_FIFOStatus.FifoPreFull
	    THEN
	        // Status
	        IF (#t_UDT_ColumnLiftStatus.Status <> #s_UDT_ColumnLiftOld.Status OR (#sx_SendAllProcedure AND #ii_ErrorNumber = 0))
	        THEN
	            #sx_ItemStatusMessageReq := TRUE;
	            #si_ItemStatus := #t_UDT_ColumnLiftStatus.Status;
	            #s_UDT_ColumnLiftOld.Status := #t_UDT_ColumnLiftStatus.Status;
	        END_IF;


	        // Check which specific status changed, prepare code, change state and write new status into the old one.
	        IF (#t_UDT_ColumnLiftStatus.Specific.ReferenceError <> #s_UDT_ColumnLiftOld.Specific.ReferenceError AND NOT #sx_SendAllProcedure)
	            OR (#sx_SendAllProcedure AND #ii_ErrorNumber = 0)
	        THEN
	            #sdi_Code := "DB_MFC_ErrorCode".ColumnLift.ReferenceError;
	            #si_State := BOOL_TO_INT(#t_UDT_ColumnLiftStatus.Specific.ReferenceError);
	            #s_UDT_ColumnLiftOld.Specific.ReferenceError := #t_UDT_ColumnLiftStatus.Specific.ReferenceError;
	            #sx_ItemErrorMessageReq := TRUE;
	            #ii_ErrorNumber += 1;
	        ELSIF (#t_UDT_ColumnLiftStatus.Specific.SwitchingTimerError <> #s_UDT_ColumnLiftOld.Specific.SwitchingTimerError AND NOT #sx_SendAllProcedure)
	            OR (#sx_SendAllProcedure AND #ii_ErrorNumber = 1)
	        THEN
	            #sdi_Code := "DB_MFC_ErrorCode".ColumnLift.SwitchingTimerError;
	            #si_State := BOOL_TO_INT(#t_UDT_ColumnLiftStatus.Specific.SwitchingTimerError);
	            #s_UDT_ColumnLiftOld.Specific.SwitchingTimerError := #t_UDT_ColumnLiftStatus.Specific.SwitchingTimerError;
	            #sx_ItemErrorMessageReq := TRUE;
	            #ii_ErrorNumber += 1;
	        ELSIF (#t_UDT_ColumnLiftStatus.Specific.LimitSensorUpperPosition <> #s_UDT_ColumnLiftOld.Specific.LimitSensorUpperPosition AND NOT #sx_SendAllProcedure)
	            OR (#sx_SendAllProcedure AND #ii_ErrorNumber = 2)
	        THEN
	            #sdi_Code := "DB_MFC_ErrorCode".ColumnLift.LimitSensorUpperPosition;
	            #si_State := BOOL_TO_INT(#t_UDT_ColumnLiftStatus.Specific.LimitSensorUpperPosition);
	            #s_UDT_ColumnLiftOld.Specific.LimitSensorUpperPosition := #t_UDT_ColumnLiftStatus.Specific.LimitSensorUpperPosition;
	            #sx_ItemErrorMessageReq := TRUE;
	            #ii_ErrorNumber += 1;
	        ELSIF (#t_UDT_ColumnLiftStatus.Specific.LimitSensorLowerPosition <> #s_UDT_ColumnLiftOld.Specific.LimitSensorLowerPosition AND NOT #sx_SendAllProcedure)
	            OR (#sx_SendAllProcedure AND #ii_ErrorNumber = 3)
	        THEN
	            #sdi_Code := "DB_MFC_ErrorCode".ColumnLift.LimitSensorLowerPosition;
	            #si_State := BOOL_TO_INT(#t_UDT_ColumnLiftStatus.Specific.LimitSensorLowerPosition);
	            #s_UDT_ColumnLiftOld.Specific.LimitSensorLowerPosition := #t_UDT_ColumnLiftStatus.Specific.LimitSensorLowerPosition;
	            #sx_ItemErrorMessageReq := TRUE;
	            #ii_ErrorNumber += 1;
	        ELSIF (#t_UDT_ColumnLiftStatus.Specific.UpperPosition <> #s_UDT_ColumnLiftOld.Specific.UpperPosition AND NOT #sx_SendAllProcedure)
	            OR (#sx_SendAllProcedure AND #ii_ErrorNumber = 4)
	        THEN
	            #sdi_Code := "DB_MFC_ErrorCode".ColumnLift.UpperPosition;
	            #si_State := BOOL_TO_INT(#t_UDT_ColumnLiftStatus.Specific.UpperPosition);
	            #s_UDT_ColumnLiftOld.Specific.UpperPosition := #t_UDT_ColumnLiftStatus.Specific.UpperPosition;
	            #sx_ItemErrorMessageReq := TRUE;
	            #ii_ErrorNumber += 1;
	        ELSIF (#t_UDT_ColumnLiftStatus.Specific.LowerPosition <> #s_UDT_ColumnLiftOld.Specific.LowerPosition AND NOT #sx_SendAllProcedure)
	            OR (#sx_SendAllProcedure AND #ii_ErrorNumber = 5)
	        THEN
	            #sdi_Code := "DB_MFC_ErrorCode".ColumnLift.LowerPosition;
	            #si_State := BOOL_TO_INT(#t_UDT_ColumnLiftStatus.Specific.LowerPosition);
	            #s_UDT_ColumnLiftOld.Specific.LowerPosition := #t_UDT_ColumnLiftStatus.Specific.LowerPosition;
	            #sx_ItemErrorMessageReq := TRUE;
	            #ii_ErrorNumber += 1;
	        ELSIF (#t_UDT_ColumnLiftStatus.Specific.ChuteNotInPosition <> #s_UDT_ColumnLiftOld.Specific.ChuteNotInPosition AND NOT #sx_SendAllProcedure)
	            OR (#sx_SendAllProcedure AND #ii_ErrorNumber = 6)
	        THEN
	            #sdi_Code := "DB_MFC_ErrorCode".ColumnLift.ChuteNotInPosition;
	            #si_State := BOOL_TO_INT(#t_UDT_ColumnLiftStatus.Specific.ChuteNotInPosition);
	            #s_UDT_ColumnLiftOld.Specific.ChuteNotInPosition := #t_UDT_ColumnLiftStatus.Specific.ChuteNotInPosition;
	            #sx_ItemErrorMessageReq := TRUE;
	            #sx_SendAllProcedure := FALSE;
	            #ii_ErrorNumber += 1;
	        END_IF;
	    END_IF;
	END_REGION

	REGION 4 - Write message components to the item error structure

	    #s_UDT_ItemError.ItemNumber := #i_UDT_EquipmentNumber;
	    #s_UDT_ItemError.Error := #sdi_Code;
	    #s_UDT_ItemError.State := #si_State;
	    #s_UDT_ItemError.Masked := 1;

	END_REGION

	REGION 5 - Write message components to the item status structure

	    #s_UDT_ItemStatus.Group := #i_UDT_EquipmentNumber.Group;
	    #s_UDT_ItemStatus.Node := #i_UDT_EquipmentNumber.Node;
	    #s_UDT_ItemStatus.Status := #si_ItemStatus;

	END_REGION

	REGION 6 - Prepare messages to the MFC

	    // If item error message required signal is set, prepare the item error message.
	    IF (#sx_ItemErrorMessageReq)
	    THEN
	        #s_FB_ItemError(i_UDT_ItemErrorBody := #s_UDT_ItemError,
	                        ii_MessageGroup := 1,
	                        ix_FlagRetry := FALSE,
	                        idi_TimeSpan := 0,
	                        qx_Error => #sx_ItemErrorBlockError,
	                        qx_Warning => #sx_ItemErrorBlockWarning,
	                        iq_UDT_FifoHeader := #iq_UDT_FifoHeader,
	                        iqs_FifoData := #iqs_FifoData,
	                        iqdi_MessageSequenceNumber := #iqdi_MessageSequenceNumber);
	    END_IF;

	    // If item status message required signal is set, prepare the item error message.
	    IF (#sx_ItemStatusMessageReq)
	    THEN
	        #s_FB_ItemStatus(i_UDT_ItemStatusBody := #s_UDT_ItemStatus,
	                         ii_MessageGroup := 1,
	                         ix_FlagRetry := FALSE,
	                         idi_TimeSpan := 0,
	                         qx_Error => #sx_ItemStatusBlockError,
	                         qx_Warning => #sx_ItemStatusBlockWarning,
	                         iq_UDT_FifoHeader := #iq_UDT_FifoHeader,
	                         iqs_FifoData := #iqs_FifoData,
	                         iqdi_MessageSequenceNumber := #iqdi_MessageSequenceNumber);
	    END_IF;

	END_REGION

	REGION 7 - Write outputs

	    // Prepare collective output error.
	    #qx_Error :=
	    #sx_ItemErrorBlockError
	    OR #sx_ItemStatusBlockError
	    OR #sx_FIFOError;

	    // Prepare collective output warning.
	    #qx_Warning :=
	    #sx_ItemErrorBlockWarning
	    OR #sx_ItemStatusBlockWarning
	    OR #sx_FIFOWarning;

	END_REGION
END_FUNCTION_BLOCK

FUNCTION_BLOCK "FB_MFC_Visu_BiDirectionalStatus"
{ S7_Optimized_Access := 'TRUE' }
VERSION : 0.1
// ATTRIBUTES
// AUTO_NUMBER = True
// BLOCK_NUMBER = 136
// END_ATTRIBUTES
   VAR_INPUT
      i_UDT_BiDirectionalStatus { ExternalAccessible := 'False'; ExternalVisible := 'False'; ExternalWritable := 'False'} : "UDT_BiDirectionalStatus";   // MCP status structure
      i_UDT_EquipmentNumber { ExternalAccessible := 'False'; ExternalVisible := 'False'; ExternalWritable := 'False'} : "UDT_EquipmentNumber";   // Item number
      ix_SendAllErrorsState { ExternalAccessible := 'False'; ExternalVisible := 'False'; ExternalWritable := 'False'} : Bool;   // True - update all the messages
      ix_MFCConnected { ExternalAccessible := 'False'; ExternalVisible := 'False'; ExternalWritable := 'False'} : Bool;   // True - A connection to the MFC has been established
      ix_CollectiveReset { ExternalAccessible := 'False'; ExternalVisible := 'False'; ExternalWritable := 'False'} : Bool;   // True - Collective reset command of all system controls
   END_VAR

   VAR_OUTPUT
      qx_Error { ExternalAccessible := 'False'; ExternalVisible := 'False'; ExternalWritable := 'False'} : Bool;   // Block error
      qx_Warning { ExternalAccessible := 'False'; ExternalVisible := 'False'; ExternalWritable := 'False'} : Bool;   // Block warning
   END_VAR

   VAR_IN_OUT
      iq_UDT_FifoHeader : "UDT_FifoHeader";   // FIFO header
      iqs_FifoData : Array[*] of "UDT_MessageV2";   // FIFO data buffer
      iqdi_MessageSequenceNumber { ExternalAccessible := 'False'; ExternalVisible := 'False'; ExternalWritable := 'False'} : DInt;   // Message number
   END_VAR

   VAR
      sx_ItemErrorMessageReq { ExternalAccessible := 'False'; ExternalVisible := 'False'; ExternalWritable := 'False'} : Bool;   // Item error message required
      sx_ItemStatusMessageReq { ExternalAccessible := 'False'; ExternalVisible := 'False'; ExternalWritable := 'False'} : Bool;   // Item status message required
      s_R_TRIG_Connection {InstructionName := 'R_TRIG'; LibVersion := '1.0'; ExternalAccessible := 'False'; ExternalVisible := 'False'; ExternalWritable := 'False'; S7_SetPoint := 'False'} : R_TRIG;   // Rising edge trigger connection reastablished
      s_F_TRIG_SendAllErrors {InstructionName := 'F_TRIG'; LibVersion := '1.0'; ExternalAccessible := 'False'; ExternalVisible := 'False'; ExternalWritable := 'False'; S7_SetPoint := 'False'} : F_TRIG;   // Falling edge trigger from signal send all errors
      si_ItemStatus { ExternalAccessible := 'False'; ExternalVisible := 'False'; ExternalWritable := 'False'} : Int;   // Item status
      sx_SendAllProcedure { ExternalAccessible := 'False'; ExternalVisible := 'False'; ExternalWritable := 'False'} : Bool;   // Send all procedure
      ii_ErrorNumber { ExternalAccessible := 'False'; ExternalVisible := 'False'; ExternalWritable := 'False'} : Int;   // Counter Error Number
      ss_FIFOStatus { ExternalAccessible := 'False'; ExternalVisible := 'False'; ExternalWritable := 'False'; S7_SetPoint := 'False'} : "UDT_FifoStatus";   // Status structure
      sx_FIFOError { ExternalAccessible := 'False'; ExternalVisible := 'False'; ExternalWritable := 'False'} : Bool;   // FIFO error
      sx_FIFOWarning { ExternalAccessible := 'False'; ExternalVisible := 'False'; ExternalWritable := 'False'} : Bool;   // FIFO warning
      s_UDT_Message { ExternalAccessible := 'False'; ExternalVisible := 'False'; ExternalWritable := 'False'; S7_SetPoint := 'False'} : "UDT_MessageV2";   // Message
      s_UDT_BiDirectionalStatusOld { ExternalAccessible := 'False'; ExternalVisible := 'False'; ExternalWritable := 'False'; S7_SetPoint := 'False'} : "UDT_BiDirectionalStatus";   // MCP old status structure
      s_UDT_ItemError { ExternalAccessible := 'False'; ExternalVisible := 'False'; ExternalWritable := 'False'; S7_SetPoint := 'False'} : "UDT_ItemError";   // Item error message body structure
      sdi_Code { ExternalAccessible := 'False'; ExternalVisible := 'False'; ExternalWritable := 'False'} : DInt;   // Error code
      si_State { ExternalAccessible := 'False'; ExternalVisible := 'False'; ExternalWritable := 'False'} : Int;   // Error state
      si_Rack { ExternalAccessible := 'False'; ExternalVisible := 'False'; ExternalWritable := 'False'} : Int;
      si_IOModule { ExternalAccessible := 'False'; ExternalVisible := 'False'; ExternalWritable := 'False'} : Int;
      s_UDT_ItemStatus { ExternalAccessible := 'False'; ExternalVisible := 'False'; ExternalWritable := 'False'; S7_SetPoint := 'False'} : "UDT_ItemStatus";   // Item status message body structure
      s_FB_ItemStatus { ExternalAccessible := 'False'; ExternalVisible := 'False'; ExternalWritable := 'False'; S7_SetPoint := 'False'} : "FB_ItemStatus";   // Item status block's instance
      s_FB_ItemError { ExternalAccessible := 'False'; ExternalVisible := 'False'; ExternalWritable := 'False'; S7_SetPoint := 'False'} : "FB_ItemError";   // Item error block's instance
      sx_ItemErrorBlockError { ExternalAccessible := 'False'; ExternalVisible := 'False'; ExternalWritable := 'False'} : Bool;   // Item error block error
      sx_ItemErrorBlockWarning { ExternalAccessible := 'False'; ExternalVisible := 'False'; ExternalWritable := 'False'} : Bool;   // Item error block warning
      sx_ItemStatusBlockError { ExternalAccessible := 'False'; ExternalVisible := 'False'; ExternalWritable := 'False'} : Bool;   // Item status block error
      sx_ItemStatusBlockWarning { ExternalAccessible := 'False'; ExternalVisible := 'False'; ExternalWritable := 'False'} : Bool;   // Item status block warning
   END_VAR


BEGIN
	(*
	----------------------------------------------------------------------------------------
	|                                                                                      |
	|  Copyright  2023             FORTNA Europe BV                                        |
	|  All Rights Reserved         Netherlands                                             |
	|                                                                                      |
	----------------------------------------------------------------------------------------
	Version history:
	Date        | Version   | Author       | Remark
	----------------------------------------------------------------------------------------
	28/03/2023  | 1.0       | M. Diebel   | Release TIA 17 | DHL Munich 2023
	13/03/2023  | 1.1       | S. Nieswiec | Updated for new Baseline
	*)


	REGION 1 - Initialize message required signals

	    #sx_ItemErrorMessageReq := FALSE;


	    // On connection reestablish send last remembered status and error state ( status only when it's diffrent then 0 )
	    #s_R_TRIG_Connection(CLK := #ix_MFCConnected);


	    IF #s_R_TRIG_Connection.Q
	    THEN
	        #sx_ItemErrorMessageReq := TRUE;
	    END_IF;

	    // Prepare trigger on the collective reset signal.
	    #s_F_TRIG_SendAllErrors(CLK := #ix_SendAllErrorsState);

	    // When collective reset will go down, start send every equipment errors.
	    IF #s_F_TRIG_SendAllErrors.Q AND NOT #sx_SendAllProcedure
	    THEN
	        #ii_ErrorNumber := 0;
	        #sx_SendAllProcedure := TRUE;
	    END_IF;

	END_REGION

	REGION 2 - FIFO header status update

	    // Mode 'S' - FIFO register status update.
	    "FC_Fifo"(ic_Mode := 'S',
	              qUDT_Status => #ss_FIFOStatus,
	              qx_Error => #sx_FIFOError,
	              qx_Warning => #sx_FIFOWarning,
	              iqv_Data := #s_UDT_Message,
	              iqUDT_FifoHeader := #iq_UDT_FifoHeader,
	              iqv_DataBuffer := #iqs_FifoData);

	END_REGION

	REGION 3 - Prepare message data

	    // When there is no reset errors command, update status and errors.
	    IF NOT #ix_CollectiveReset
	        AND NOT #ss_FIFOStatus.FifoPreFull
	    THEN

	        // Check which specific status changed, prepare code, change state and write new status into the old one.
	        IF (#i_UDT_BiDirectionalStatus.InfeedModeRequested <> #s_UDT_BiDirectionalStatusOld.InfeedModeRequested AND NOT #sx_SendAllProcedure)
	            OR (#sx_SendAllProcedure AND #ii_ErrorNumber = 0)
	        THEN
	            #sdi_Code := "DB_MFC_ErrorCode".BiDirectional.InfeedModeRequested;
	            #si_State := BOOL_TO_INT(#i_UDT_BiDirectionalStatus.InfeedModeRequested);
	            #s_UDT_BiDirectionalStatusOld.InfeedModeRequested := #i_UDT_BiDirectionalStatus.InfeedModeRequested;
	            #sx_ItemErrorMessageReq := TRUE;
	            #ii_ErrorNumber += 1;
	        ELSIF (#i_UDT_BiDirectionalStatus.OutfeedModeRequested <> #s_UDT_BiDirectionalStatusOld.OutfeedModeRequested AND NOT #sx_SendAllProcedure)
	            OR (#sx_SendAllProcedure AND #ii_ErrorNumber = 1)
	        THEN
	            #sdi_Code := "DB_MFC_ErrorCode".BiDirectional.OutfeedModeRequested;
	            #si_State := BOOL_TO_INT(#i_UDT_BiDirectionalStatus.OutfeedModeRequested);
	            #s_UDT_BiDirectionalStatusOld.OutfeedModeRequested := #i_UDT_BiDirectionalStatus.OutfeedModeRequested;
	            #sx_ItemErrorMessageReq := TRUE;
	            #ii_ErrorNumber += 1;
	        ELSIF (#i_UDT_BiDirectionalStatus.InfeedModeActive <> #s_UDT_BiDirectionalStatusOld.InfeedModeActive AND NOT #sx_SendAllProcedure)
	            OR (#sx_SendAllProcedure AND #ii_ErrorNumber = 2)
	        THEN
	            #sdi_Code := "DB_MFC_ErrorCode".BiDirectional.InfeedModeActive;
	            #si_State := BOOL_TO_INT(#i_UDT_BiDirectionalStatus.InfeedModeActive);
	            #s_UDT_BiDirectionalStatusOld.InfeedModeActive := #i_UDT_BiDirectionalStatus.InfeedModeActive;
	            #sx_ItemErrorMessageReq := TRUE;
	            #ii_ErrorNumber += 1;
	        ELSIF (#i_UDT_BiDirectionalStatus.OutfeedModeActive <> #s_UDT_BiDirectionalStatusOld.OutfeedModeActive AND NOT #sx_SendAllProcedure)
	            OR (#sx_SendAllProcedure AND #ii_ErrorNumber = 3)
	        THEN
	            #sdi_Code := "DB_MFC_ErrorCode".BiDirectional.OutfeedModeActive;
	            #si_State := BOOL_TO_INT(#i_UDT_BiDirectionalStatus.OutfeedModeActive);
	            #s_UDT_BiDirectionalStatusOld.OutfeedModeActive := #i_UDT_BiDirectionalStatus.OutfeedModeActive;
	            #sx_ItemErrorMessageReq := TRUE;
	            #ii_ErrorNumber += 1;
	        ELSIF (#i_UDT_BiDirectionalStatus.InfeedModeReady <> #s_UDT_BiDirectionalStatusOld.InfeedModeReady AND NOT #sx_SendAllProcedure)
	            OR (#sx_SendAllProcedure AND #ii_ErrorNumber = 4)
	        THEN
	            #sdi_Code := "DB_MFC_ErrorCode".BiDirectional.InfeedModeReady;
	            #si_State := BOOL_TO_INT(#i_UDT_BiDirectionalStatus.InfeedModeReady);
	            #s_UDT_BiDirectionalStatusOld.InfeedModeReady := #i_UDT_BiDirectionalStatus.InfeedModeReady;
	            #sx_ItemErrorMessageReq := TRUE;
	            #ii_ErrorNumber += 1;
	        ELSIF (#i_UDT_BiDirectionalStatus.OutfeedModeReady <> #s_UDT_BiDirectionalStatusOld.OutfeedModeReady AND NOT #sx_SendAllProcedure)
	            OR (#sx_SendAllProcedure AND #ii_ErrorNumber = 5)
	        THEN
	            #sdi_Code := "DB_MFC_ErrorCode".BiDirectional.OutfeedModeReady;
	            #si_State := BOOL_TO_INT(#i_UDT_BiDirectionalStatus.OutfeedModeReady);
	            #s_UDT_BiDirectionalStatusOld.OutfeedModeReady := #i_UDT_BiDirectionalStatus.OutfeedModeReady;
	            #sx_ItemErrorMessageReq := TRUE;
	            #ii_ErrorNumber += 1;
	            #sx_SendAllProcedure := FALSE;
	        END_IF;
	    END_IF;
	END_REGION

	REGION 4 - Write message components to the item error structure

	    #s_UDT_ItemError.ItemNumber := #i_UDT_EquipmentNumber;
	    #s_UDT_ItemError.Error := #sdi_Code;
	    #s_UDT_ItemError.State := #si_State;
	    #s_UDT_ItemError.Masked := 1;

	END_REGION



	REGION 5 - Prepare messages to the MFC

	    // If item error message required signal is set, prepare the item error message.
	    IF (#sx_ItemErrorMessageReq)
	    THEN
	        #s_FB_ItemError(i_UDT_ItemErrorBody := #s_UDT_ItemError,
	                        ii_MessageGroup := 1,
	                        ix_FlagRetry := FALSE,
	                        idi_TimeSpan := 0,
	                        qx_Error => #sx_ItemErrorBlockError,
	                        qx_Warning => #sx_ItemErrorBlockWarning,
	                        iq_UDT_FifoHeader := #iq_UDT_FifoHeader,
	                        iqs_FifoData := #iqs_FifoData,
	                        iqdi_MessageSequenceNumber := #iqdi_MessageSequenceNumber);
	    END_IF;


	END_REGION

	REGION 7 - Write outputs

	    // Prepare collective output error.
	    #qx_Error :=
	    #sx_ItemErrorBlockError
	    OR #sx_FIFOError;

	    // Prepare collective output warning.
	    #qx_Warning :=
	    #sx_ItemErrorBlockWarning
	    OR #sx_FIFOWarning;

	END_REGION
END_FUNCTION_BLOCK

FUNCTION_BLOCK "FB_MFC_Visu_CodingBeltModes_Status"
{ S7_Optimized_Access := 'TRUE' }
VERSION : 1.1
// ATTRIBUTES
// AUTO_NUMBER = True
// BLOCK_NUMBER = 138
// END_ATTRIBUTES
   VAR_INPUT
      i_UDT_CodingBeltModesStatus { ExternalAccessible := 'False'; ExternalVisible := 'False'; ExternalWritable := 'False'} : "UDT_CodingBeltModesStatus";   // CodingBeltModes status structure
      i_UDT_EquipmentNumber { ExternalAccessible := 'False'; ExternalVisible := 'False'; ExternalWritable := 'False'} : "UDT_EquipmentNumber";   // Item number
      ix_SendAllErrorsState { ExternalAccessible := 'False'; ExternalVisible := 'False'; ExternalWritable := 'False'} : Bool;   // True - update all the messages
      ix_MFCConnected { ExternalAccessible := 'False'; ExternalVisible := 'False'; ExternalWritable := 'False'} : Bool;   // True - A connection to the MFC has been established
      ix_CollectiveReset { ExternalAccessible := 'False'; ExternalVisible := 'False'; ExternalWritable := 'False'} : Bool;   // True - Collective reset command of all system controls
   END_VAR

   VAR_OUTPUT
      qx_Error { ExternalAccessible := 'False'; ExternalVisible := 'False'; ExternalWritable := 'False'} : Bool;   // Block error
      qx_Warning { ExternalAccessible := 'False'; ExternalVisible := 'False'; ExternalWritable := 'False'} : Bool;   // Block warning
   END_VAR

   VAR_IN_OUT
      iq_UDT_FifoHeader : "UDT_FifoHeader";   // FIFO header
      iqs_FifoData : Array[*] of "UDT_MessageV2";   // FIFO data buffer
      iqdi_MessageSequenceNumber { ExternalAccessible := 'False'; ExternalVisible := 'False'; ExternalWritable := 'False'} : DInt;   // Message number
   END_VAR

